(* IEC 61131-3 sources: beebread/doc (part 6) *)

// Commented out for beedance: it uses CODE, which is commented out.
// FUNCTION_BLOCK DNS_REV_CLIENT
// VAR_IN_OUT
// 	IP_C : IP_C; (* IP_Control management structure *)
// 	S_BUF : NETWORK_BUFFER;
// 	R_BUF : NETWORK_BUFFER;
// END_VAR
// VAR_INPUT
// 	ACTIVATE : BOOL;
// 	IP4 : DWORD;
// 	IP4_DNS : DWORD;
// END_VAR
// VAR_OUTPUT
// 	DOMAIN : STRING;
// 	DONE : BOOL;
// 	ERROR : DWORD;
// END_VAR
// VAR
// 	IP_FIFO : IP_FIFO;
// 	ip_state : BYTE;
// 	ip_id : BYTE;
// 	state : INT;
// 	ip4_copy : DWORD;
// 	d : STRING(27);
// 	activate_last : BOOL;
// 	i : INT;
// 	dl : INT;
// 	p1 : INT;
// 	char : BYTE;
// 	char_count : INT;
// 	tid : BYTE;
// END_VAR
//
// (* Domain Name System (query) *)
//
// CASE state OF
// 00: (* wait for rising edge on GET *)
// 	IF ACTIVATE AND NOT activate_last THEN
// 		ERROR := DWORD#0;
// 		ip4_copy := ip4; (* save IP4 *)
// 		ip_state := BYTE#1;
// 		DOMAIN := '';
// 		DONE := FALSE;
//
// 		d := '';
// 		FOR i := 1 TO 4 DO
// 			d := CONCAT(d,BYTE_TO_STRING(DWORD_TO_BYTE(IP4)));
// 			d := CONCAT(d,'.');
// 			IP4 := ROR(IP4,8);
// 		END_FOR;
// 		d := CONCAT(d,'in-addr.arpa');
// 		state := 10;
// 	END_IF;
//
// 10: (* register with IP_Control *)
// 	IF ip_state = BYTE#3 THEN
// 		dl := LEN(d);
//
// 		(* initialize send buffer *)
// 		char_count := 17 + dl;
// 		FOR i := 0 TO char_count DO
// 			S_BUF.BUFFER[i] := BYTE#00;
// 		END_FOR;
//
// 		tid := UINT_TO_BYTE(BYTE_TO_UINT(tid) + UINT#1);
// 		S_BUF.BUFFER[01] := tid; (* Transaction ID lowbyte *)
// 		S_BUF.BUFFER[02] := BYTE#16#01; (* Flags: highbyte *)
// 		S_BUF.BUFFER[05] := BYTE#16#01; (* Questions: lowbyte *)
//
// 		(* process the server name from back to front *)
// 		i := dl + 12;
// 		char_count := 0;
//
// 		WHILE i > 12 DO
// 			char := CODE(STR:=d,POS:=i - 12);
//
// 			(* check for main/sub domain name separator "." *)
// 			IF char = BYTE#46 THEN
// 				(* instead of the separator "." the length of the detected main/sub domain name is entered *)
// 				S_BUF.BUFFER[i] := INT_TO_BYTE(char_count);
// 				char_count := 0;
// 			ELSE
// 				S_BUF.BUFFER[i] := char; (* enter char into buffer *)
// 				char_count := char_count + 1; (* count number of chars *)
// 			END_IF;
// 			i := i - 1;
// 		END_WHILE;
//
// 		S_BUF.BUFFER[i] := INT_TO_BYTE(char_count); (* enter the length of the leftmost (first) domain name *)
// 		i := dl + 15; (* position after the server name *)
// 		S_BUF.BUFFER[i] := BYTE#12; (* Type: PTR (Domain name pointer) lowbyte *)
// 		i := i + 2;
// 		S_BUF.BUFFER[i] := BYTE#01; (* Class: IN lowbyte *)
// 		i := i + 1;
//
// 		(* set up IP data traffic *)
// 		IP_C.C_PORT := WORD#53; (* enter port number *)
// 		IP_C.C_IP := IP4_DNS; (* enter IP *)
// 		IP_C.C_MODE := BYTE#1; (* Mode: UDP+ACTIVE+PORT+IP *)
// 		IP_C.C_ENABLE := TRUE; (* enable connection setup *)
// 		IP_C.TIME_RESET := TRUE; (* reset timeout monitoring *)
// 		IP_C.R_OBSERVE  := TRUE; (* monitor data reception *)
// 		S_BUF.SIZE := INT_TO_UINT(i); (* enter send length *)
// 		R_BUF.SIZE := UINT#0; (* reset receive length *)
// 		state := 30;
// 	END_IF;
//
// 30:
// 	IF IP_C.ERROR <> DWORD#00 THEN
// 		ERROR := IP_C.ERROR;
// 	(* check whether the response telegram has the correct transaction ID and minimum length *)
// 	ELSIF (S_BUF.SIZE = UINT#0) AND (tid = R_BUF.BUFFER[1]) AND (R_BUF.SIZE >= INT_TO_UINT(i+12)) THEN
//
// 		(* check return code of the flags. 4 bits *)
// 		ERROR := BYTE_TO_DWORD(R_BUF.BUFFER[3] AND BYTE#2#0000_1111);
//
// 		IF ERROR = DWORD#00 THEN
//
// 			i := R_BUF.SIZE - 2;
// 			WHILE R_BUF.BUFFER[i] > 0 DO
// 				IF i = 0 THEN EXIT; END_IF;
// 				i := i - 1;
// 			END_WHILE;
//
// 			i := i + 2;
// 			p1 := i + 1;
// 			WHILE i < R_BUF.SIZE DO
// 				dl := R_BUF.BUFFER[i];
// 				IF dl > 0 THEN
// 					R_BUF.BUFFER[i] := BYTE#46;
// 					i := i + dl + 1;
// 				ELSE
// 					DOMAIN := BUFFER_TO_STRING(PT:=REF(R_BUF.BUFFER),SIZE:=SIZEOF(R_BUF.BUFFER),START:=p1,STOP:=i-1);
// 					EXIT;
// 				END_IF;
// 			END_WHILE;
// 			state := 0;
// 			DONE := TRUE;
// 		END_IF;
// 	END_IF;
//
// 	IF ERROR <> DWORD#0 THEN
// 		state := 0;
// 	END_IF;
//
// 	IF state = 0 THEN
// 		IP_C.R_OBSERVE := FALSE; (* monitor data reception *)
// 		ip_state := BYTE#4; (* unregister *)
// 	END_IF;
//
// END_CASE;
//
// activate_last := ACTIVATE; (* save last status for edge detection *)
//
// (* IP_FIFO *)
// IP_FIFO(FIFO:=IP_C.FIFO,STATE:=ip_state,ID:=ip_id);
//
// (*----------------------------------------------------------------------------------------------------------------*)
// (* Flags: 0x0100 (Standard query)                                                                                            *)
// (* 0... .... .... .... = Response: Message is a query                                                                   *)
// (* .000 0... ....  = Opcode: Standard query (0)                                                                          *)
// (* .... ..0. .... .... = Truncated: Message is not truncated                                                          *)
// (* .... ...1 .... .... = Recursion desired: Do query recursively                                                    *)
// (* .... .... .0.. .... = Z: reserved (0)                                                                                                  *)
// (* .... .... ...0 .... = Non-authenticated data OK: Non-authenticated data is unacceptable *)
// (*-----------------------------------------------------------------------------------------------------------------*)
//
// (*
// Errorcodes  Description	References
// 000	No error. 		 	The request completed successfully.
// 001	Format error. 		The name server was unable to interpret the query.
// 002	Server failure.  	The name server was unable to process this query due to a problem with the name server.
// 003	Name Error. 	 	Meaningful only for responses from an authoritative name server, this code signifies that the domain name referenced in the query does not exist.
// 004	Not Implemented. 	The name server does not support the requested kind of query.
// 005	Refused. 			The name server refuses to perform the specified operation for policy reasons.
//   						 For example, a name server may not wish to provide the information to the particular requester, or a name server may not wish to perform a particular operation (e.g., zone transfer) for particular data.
// 006	YXDomain.			Name Exists when it should not.
// 007	YXRRSet. RR			Set Exists when it should not.
// 008	NXRRSet. RR			Set that should exist does not.
// 009	NotAuth.			Server Not Authoritative for zone.
// 010	NotZone,			Name not contained in zone.
// 255	Timeout				No Response
// *)
// END_FUNCTION_BLOCK

// Commented out for beedance: it reads or writes the bytes of a STRING through a pointer; a beedance reference (REF_TO) refers to a whole variable of its type.
// FUNCTION ELEMENT_COUNT : INT
// VAR_INPUT
// 	SEP : BYTE;
// END_VAR
// VAR_IN_OUT
// 	ELEMENT : STRING(ELEMENT_LENGTH);
// END_VAR
// VAR
// 	pt : REF_TO ARRAY[1..ELEMENT_LENGTH] OF BYTE;
// 	l: INT;
// 	pos: INT;
// END_VAR
//
// IF ELEMENT = '' THEN
// 	ELEMENT_COUNT := 0;
// ELSE
// 	PT := REF(ELEMENT);
// 	ELEMENT_COUNT := 1;
// 	l := LEN(ELEMENT);
// 	FOR pos := 1 TO l DO
// 		IF pt^[pos] = SEP THEN ELEMENT_COUNT := ELEMENT_COUNT + 1; END_IF;
// 	END_FOR;
// END_IF;
// END_FUNCTION

// Commented out for beedance: it reads or writes the bytes of a STRING through a pointer; a beedance reference (REF_TO) refers to a whole variable of its type.
// FUNCTION ELEMENT_GET : STRING(ELEMENT_LENGTH)
// VAR_INPUT
// 	SEP : BYTE;
// 	POS : INT;
// END_VAR
// VAR_IN_OUT
// 	ELEMENT : STRING(ELEMENT_LENGTH);
// END_VAR
// VAR
// 	i : INT := 1;
// 	o : INT := 1;
// 	pt : REF_TO ARRAY[1..ELEMENT_LENGTH] OF BYTE;
// 	po : REF_TO ARRAY[1..ELEMENT_LENGTH] OF BYTE;
// 	cnt: INT;
// 	c: BYTE;
// END_VAR
//
// (* load pointers *)
// pt := REF(ELEMENT);
// po := REF(ELEMENT_GET);
//
// (* search for the n-th occurence of a separation character and store position in i *)
// WHILE (cnt < pos) AND (i < ELEMENT_LENGTH) AND (pt^[i] > 0) DO
// 	IF pt^[i] = sep THEN cnt := cnt + 1; END_IF;
// 	i := i + 1;
// END_WHILE;
//
// (* copy the list element to output *)
// IF i < ELEMENT_LENGTH THEN c := pt^[i]; END_IF;
// WHILE (c <> sep) AND (c > 0) AND (o < ELEMENT_LENGTH) AND (i < ELEMENT_LENGTH) DO
// 	po^[o] :=pt^[i];
// 	o := o + 1;
// 	i := i + 1;
// 	c := pt^[i];
// END_WHILE;
//
// (* terminate the output string *)
// po^[o] := 0;
// END_FUNCTION

FUNCTION_BLOCK FILE_BLOCK
VAR_IN_OUT
	MODE : BYTE;
	FILENAME : STRING;
	FSD : FILE_SERVER_DATA;
	PT : NETWORK_BUFFER;
END_VAR
VAR_INPUT
	POS : UDINT;
END_VAR
VAR_OUTPUT
	ERROR : BYTE;
	DATA : BYTE;
END_VAR
VAR
	step : INT;
	i : INT;
	data_start : UDINT;
	data_stop : UDINT;

END_VAR

CASE step OF
0:	IF MODE > 0 THEN
		ERROR := 0;
		IF FSD.FILE_OPEN AND (FSD.FILE_SIZE = 0 OR POS >= FSD.FILE_SIZE) THEN
			ERROR := 255;
			MODE := 0;
		ELSIF POS < data_start OR POS > data_stop OR NOT FSD.FILE_OPEN THEN (* reading data necessary *)
			FSD.FILENAME := FILENAME;
			FSD.MODE := 1; (* open + read *)
			FSD.OFFSET := POS;
			PT.SIZE := 65535; (* read maximum number *);
			data_start := 0;
			data_stop := 0;
			step := 10;
		ELSE (* data is present in the buffer *)
			i := UDINT_TO_INT(POS - data_start); (* calculate index *)
			DATA := PT.BUFFER[i];
			MODE := 0;
			(* ---------------------- Debug-Message ----------------------------*)
			(* -----------------------------------------------------------------*)
		END_IF;
	END_IF;

10:	IF FSD.MODE = 0 THEN (* command finished *)
		IF FSD.ERROR > 0 THEN
			ERROR := FSD.ERROR; (* output error *)
			MODE := 0;
		ELSE
			data_start := POS;
			data_stop := POS + UINT_TO_UDINT(PT.SIZE) - 1;
		END_IF;
		step := 0;
	END_IF;
END_CASE;
END_FUNCTION_BLOCK

FUNCTION FILE_PATH_SPLIT : BOOL
VAR_INPUT
	FILENAME : STRING(STRING_LENGTH);
END_VAR
VAR_IN_OUT
	X : FILE_PATH_DATA;
END_VAR
VAR
	b : INT;
	c : INT;
	d : STRING(1);
	p1 : INT;
	p2 : INT;
END_VAR

X.DRIVE := '';
X.DIRECTORY := '';
X.FILENAME := '';
c := LEN(FILENAME);
IF c = 0 THEN
	FILE_PATH_SPLIT := FALSE;
	RETURN;
END_IF;

FOR b := 1 TO c DO
	d := MID(FILENAME, 1, b);
	IF d = ':' THEN
		p1 := b;
	ELSIF d = '/' OR d = '\' THEN
		p2 := b;
	END_IF;
END_FOR;

IF p1 = 2 THEN
	X.DRIVE := LEFT(FILENAME,p1);
END_IF;

IF p2 > 0 AND p2 > p1 THEN
	X.DIRECTORY := MID(FILENAME,p2 - p1,p1+1); (* len , pos *)
END_IF;

X.FILENAME := RIGHT(FILENAME,c - MAX (p1,p2));
FILE_PATH_SPLIT := TRUE;
END_FUNCTION

FUNCTION_BLOCK FILE_SERVER
VAR_IN_OUT
	FSD : FILE_SERVER_DATA;
	PT : NETWORK_BUFFER;
END_VAR
VAR
	buf_size : UDINT;
	handle : UINT; (* Filehandle *)
	read_max_length : UDINT;(* maximum data length *)
	file_position : UDINT;(* current write/read pointer *)
	used_filename : STRING;(* current file name *)
	length_read : UDINT;
	write_length : UDINT;
	length_written : UDINT;
	open_handle : UINT;
	seek_position : UDINT;
	seek_mode : INT;
	seek_data : ARRAY[0..1] OF DINT;
	tell_position : UDINT;
	open_mode : DWORD;
	last_mode: BYTE;
	command : BYTE;
	error_code : BYTE;
	error : BOOL;
	file_change : BOOL;
	step : INT;
	X : FW_AdsRdWrt;
	tmpDW : UDINT;
	para : BOOL;
	FSR : FILE_SERVER_RUNTIME;

END_VAR

CASE step OF
0:
	IF FSD.MODE = LIMIT(1,FSD.MODE,5) THEN

		(* ---------------------- Debug-Message ----------------------------*)
		(* -----------------------------------------------------------------------------*)

		(* initialization *)
		X.sNetId := '';
		X.tTimeout := T#5s;
		X.nPort := 10000; (* AMSPORT_R3_SYSSERV *)

		buf_size := SIZEOF(PT.BUFFER);

		IF FSD.MODE = 4 THEN (* File_Remove *)
			IF handle > 0 THEN
				File_change := TRUE;
				step := 32000; (* execute File_Close *)
			ELSE
				step := 90; (* execute File_Remove *)
			END_IF;

		ELSIF FSD.MODE = 5 THEN (* File_Close *)
			step := 32000; (* execute File_Close *)

		ELSIF handle = 0 THEN (* MODE 1,2,3 *)
			step := 100; (* file must be opened first *)

		ELSE (* file is open *)
			IF used_filename = FSD.FILENAME AND FSD.MODE = last_mode THEN (* no mode change? *)
				step := 200; (* continue without open procedure *)
			ELSE
				step := 32000;
				File_change := TRUE;
			END_IF;
		END_IF;
	END_IF;

(* ----------------------------------- *)
090: (* File_Remove *)
	command := 7; (* File Remove *)
	step := 95;

095: (* File_Remove finished *)
	IF command = 0 THEN
		step := 30000; (* exit *)
	END_IF;
(* ----------------------------------- *)

100: (* File_Open *)
	IF FSD.MODE = 3 THEN (* Open_New + File Write *)
		open_mode := 16#0001_001A; (* PATH_GENERIC + WRITEPLUS + BINARY *)
	ELSE (* Mode 1 Open_Exist + File _Read / Mode 2 Open_Exist + File_Write *)
		open_mode := 16#0001_0019; (* PATH_GENERIC + READPLUS + BINARY *)
	END_IF;
	command := 1; (* FileOpen *)
	step := 105;

105: (* file open finished *)
	IF command = 0 THEN
		IF error THEN
			step := 30000; (* exit *)
		ELSE
			(* enter file data *)
			handle := open_handle;
			used_filename := FSD.FILENAME;
			file_position := UDINT#4294967295; (* 16#FFFF_FFFF -> maximum = unknown *)
			last_mode := FSD.MODE;
			step := 110;
		END_IF;
	END_IF;

110: (* File Seek *)
	command := 5; (* File-Seek *)
	seek_position := 0;
	seek_mode := 2; (* SEEK_END - Seek from the end of file *)
	step := 115;

115: (* file seek finished *)
	IF command = 0 THEN
		IF error THEN
			step := 30000; (* exit *)
		ELSE
			command := 6; (* start file tell *)
			step := 120;
		END_IF;
	END_IF;

120: (* file tell finished *)
	IF command = 0 THEN
		IF error THEN
			step := 30000; (* exit *)
		ELSE
			FSD.FILE_SIZE := tell_position; (* current file size *)
			FSD.FILE_OPEN := TRUE;
			step := 200;
		END_IF;
	END_IF;

200: (* File Seek *)
	IF FSD.OFFSET = UDINT#4294967294 THEN (* 16#FFFF_FFFE -> set pointer to end of file *)
		command := 5; (* File-Seek *)
		seek_position := FSD.FILE_SIZE;
		seek_mode := 0; (* Seek from beginning of file *)
		step := 210;
	ELSIF FSD.OFFSET > FSD.FILE_SIZE THEN (* check for valid offset setting *)
		error_code := 255;
		step := 30000; (* exit *)
	ELSIF FSD.OFFSET <> file_position THEN
		command := 5; (* File-Seek *)
		seek_position := FSD.OFFSET;
		seek_mode := 0; (* Seek from beginning of file *)
		step := 210;
	ELSE
		step := 300;
	END_IF;

210: (* File Seek *)
	IF command = 0 THEN
		file_position := seek_position;
		IF error THEN
			step := 30000; (* exit *)
		ELSE
			step := 300;
		END_IF;
	END_IF;

300: (* Read or Write ? *)
	IF FSD.MODE = 1 THEN
		step := 400; (* Read *)
	ELSE
		step := 500; (* Write *)
	END_IF;

400: (* File Read *)
	IF UINT_TO_UDINT(PT.SIZE) > buf_size THEN (* limit read length to buffer size *)
		read_max_length := buf_size;
	ELSE
		read_max_length := UINT_TO_UDINT(PT.SIZE);
	END_IF;

	IF read_max_length > buf_size THEN
		read_max_length := buf_size;  (* limit read length to buffer size *)
	END_IF;

	(* adjust read length to file length *)
	IF file_position + read_max_length > FSD.FILE_SIZE THEN
		read_max_length := FSD.FILE_SIZE - file_position;
	END_IF;

	IF read_max_length > 0 THEN
		command := 3; (* File_Read *)
		step := 410;
	ELSE
		PT.SIZE := UINT#0;
		step := 30000; (* exit *)
	END_IF;

410: (* File Read *)
	IF command = 0 THEN
		PT.SIZE := UDINT_TO_UINT(length_read);
		IF NOT Error THEN
			file_position := file_position + length_read; (* correct current File_Position *)
			FSD.OFFSET := file_position;
		END_IF;
		step := 30000; (* exit *)
	END_IF;

500: (* File Write *)
	IF UINT_TO_UDINT(PT.SIZE) > buf_size THEN (* limit write length to buffer size *)
		write_length := buf_size;
	ELSE
		write_length := UINT_TO_UDINT(PT.SIZE);
	END_IF;

	IF write_length > 0 THEN
		command := 4; (* File_Write *)
		step := 510;
	ELSE
		step := 30000; (* exit *)
	END_IF;

510:
	IF command = 0 THEN
		IF NOT Error THEN
			file_position := file_position + length_written; (* correct current File_Position *)
			FSD.OFFSET := file_position;
			IF file_position > FSD.FILE_SIZE THEN (* file has grown *)
				FSD.FILE_SIZE := file_position;
			END_IF;
		END_IF;
		step := 30000; (* exit *)
	END_IF;

 (* --------------------------------------------- *)

30000: (* command done *)
	FSD.MODE := 0;
	FSD.ERROR := error_code;
	step := 0;

	(* ---------------- Debug-Message -----------------------*)
	(* --------------------------------------------- *)

32000:
	IF handle > 0 THEN
		command := 2; (* execute File_Close *)
	END_IF;
	step := 32100;

32100:
	IF command = 0 THEN (* file close finished *)
		(* clear file data *)
		FSD.FILE_OPEN := FALSE;
		file_position := 0;
		FSD.FILE_SIZE := 0;
		FSD.OFFSET := 0;
		used_filename := '';
		handle := 0;

		(* File_Name changed on the fly? *)
		IF file_change THEN
			file_change := FALSE;
			step := 0;
		ELSE
			step := 30000;
		END_IF;
	END_IF;

END_CASE;

X(bExecute := FALSE); (* cyclic FW_AdsRdWrt call *)

FSR(MODE:=BYTE#0,COMMAND:=command,FSD:=FSD); (* monitor file server runtime / command start *)

(* ------------ File Open ------------- *)
IF command = 1 THEN
	IF NOT para THEN
		para := TRUE;
		X(	nIdxGrp := 120, (* SYSTEMSERVICE_FOPEN *)
			nidxOffs := open_mode,
			cbWriteLen := SIZEOF(FSD.FILENAME),
			pWriteBuff := REF(FSD.FILENAME),
			cbReadLen := SIZEOF(tmpDW),
			pReadBuff := REF(tmpDW),
			bExecute := TRUE
			);
	ELSIF X.bBusy = FALSE THEN
		para := FALSE;
		error := X.bError;
		error_code := SEL(error,0,UDINT_TO_BYTE(X.nErrId + 16#10));

		IF X.cbRead >= SIZEOF(tmpDW) THEN
			open_handle := UDINT_TO_UINT(tmpDW);
		ELSE
			open_handle := 0;
		END_IF;
		command := 0;
		FSR(MODE:=BYTE#1,COMMAND:=command,FSD:=FSD); (* monitor file server runtime / command stop *)
		(* ---------------- Debug-Message -----------------------*)
		(* -----------------------------------------------------------------*)
	END_IF;
END_IF;

(* ----------- File Close ------------- *)
IF command = 2 THEN
	IF NOT para THEN
		para := TRUE;
		X(	nIdxGrp := 121, (* SYSTEMSERVICE_FCLOSE *)
			nidxOffs := handle,
			cbWriteLen := 0,
			pWriteBuff := 0,
			cbReadLen := 0,
			pReadBuff := 0,
			bExecute := TRUE
			);
	ELSIF X.bBusy = FALSE THEN
		para := FALSE;
		error := X.bError;
		error_code := SEL(error,0,UDINT_TO_BYTE(X.nErrId + 16#30));
		command := 0;
		FSR(MODE:=BYTE#1,COMMAND:=command,FSD:=FSD); (* monitor file server runtime / command stop *)
		(* ---------------- Debug-Message -----------------------*)
		(* -----------------------------------------------------------------*)
	END_IF;
END_IF;

(* ------------ File Read ------------- *)
IF command = 3 THEN
	IF NOT para THEN
		para := TRUE;
		X(	nIdxGrp := 122, (* SYSTEMSERVICE_FREAD *)
			nidxOffs := handle,
			cbWriteLen := 0,
			pWriteBuff := 0,
			cbReadLen := read_max_length,
			pReadBuff := REF(PT.BUFFER),
			bExecute := TRUE
			);
	ELSIF X.bBusy = FALSE THEN
		length_read := X.cbRead;
		para := FALSE;
		error := X.bError;
		error_code := SEL(error,0,UDINT_TO_BYTE(X.nErrId + 16#40));
		command := 0;
		FSR(MODE:=BYTE#1,COMMAND:=command,FSD:=FSD); (* monitor file server runtime / command stop *)
		(* ---------------- Debug-Message -----------------------*)
		(* -----------------------------------------------------------------*)
	END_IF;
END_IF;

(* ------------ File Write ------------- *)
IF command = 4 THEN
	IF NOT para THEN
		para := TRUE;
		X(	nIdxGrp := 123, (* SYSTEMSERVICE_FWRITE *)
			nidxOffs := handle,
			cbWriteLen := write_length,
			pWriteBuff := REF(PT.BUFFER),
			cbReadLen := SIZEOF(length_written),
			pReadBuff := REF(length_written),
			bExecute := TRUE
			);
	ELSIF X.bBusy = FALSE THEN
		para := FALSE;
		error := X.bError;
		error_code := SEL(error,0,UDINT_TO_BYTE(X.nErrId + 16#50));
		command := 0;
		FSR(MODE:=BYTE#1,COMMAND:=command,FSD:=FSD); (* monitor file server runtime / command stop *)
		(* ---------------- Debug-Message -----------------------*)
		(* -----------------------------------------------------------------*)
	END_IF;
END_IF;

(* ------------ File Seek ------------- *)
IF command = 5 THEN
	IF NOT para THEN
		para := TRUE;
		seek_data[0] := UDINT_TO_DINT(seek_position);
		seek_data[1] := INT_TO_DINT(seek_mode);

		X(	nIdxGrp := 124, (* SYSTEMSERVICE_FSEEK *)
			nidxOffs := handle,
			cbWriteLen := SIZEOF(seek_data),
			pWriteBuff := REF(seek_data),
			cbReadLen := 0,
			pReadBuff := 0,
			bExecute := TRUE
			);
	ELSIF X.bBusy = FALSE THEN
		para := FALSE;
		error := X.bError;
		error_code := SEL(error,0,UDINT_TO_BYTE(X.nErrId + 16#60));
		command := 0;
		FSR(MODE:=BYTE#1,COMMAND:=command,FSD:=FSD); (* monitor file server runtime / command stop *)
		(* ---------------- Debug-Message -----------------------*)
		(* -----------------------------------------------------------------*)
	END_IF;
END_IF;

(* ------------ File Tell ------------- *)
IF command = 6 THEN
	IF NOT para THEN
		para := TRUE;
		X(	nIdxGrp := 125, (* SYSTEMSERVICE_FTELL *)
			nidxOffs := handle,
			cbWriteLen := 0,
			pWriteBuff := 0,
			cbReadLen := SIZEOF(tell_position),
			pReadBuff := REF(tell_position),
			bExecute := TRUE
			);
	ELSIF X.bBusy = FALSE THEN
		para := FALSE;
		error := X.bError;
		error_code := SEL(error,0,UDINT_TO_BYTE(X.nErrId + 16#70));
		command := 0;
		FSR(MODE:=BYTE#1,COMMAND:=command,FSD:=FSD); (* monitor file server runtime / command stop *)
		(* ---------------- Debug-Message -----------------------*)
		(* -----------------------------------------------------------------*)
	END_IF;
END_IF;

(* ------------ File Remove ------------- *)
IF command = 7 THEN
	IF NOT para THEN
		para := TRUE;
		X(	nIdxGrp := 131, (* SYSTEMSERVICE_FDELETE *)
			nidxOffs := 16#0001_0000, (* PATH_GENERIC *)
			cbWriteLen := SIZEOF(FSD.FILENAME),
			pWriteBuff := REF(FSD.FILENAME),
			cbReadLen := 0,
			pReadBuff := 0,
			bExecute := TRUE
			);
	ELSIF X.bBusy = FALSE THEN
		para := FALSE;
		error := X.bError;
		error_code := SEL(error,0,UDINT_TO_BYTE(X.nErrId + 16#80));
		command := 0;
		FSR(MODE:=BYTE#1,COMMAND:=command,FSD:=FSD); (* monitor file server runtime / command stop *)
		(* ---------------- Debug-Message -----------------------*)
		(* -----------------------------------------------------------------*)
	END_IF;
END_IF;

(* ---------------- Debug-Message -----------------------*)
(* -----------------------------------------------------------------*)
END_FUNCTION_BLOCK

FUNCTION_BLOCK FILE_SERVER_RUNTIME
VAR_INPUT
	MODE : BYTE;
	COMMAND : BYTE;
END_VAR
VAR_IN_OUT
	FSD : FILE_SERVER_DATA;
END_VAR
VAR
	last_command : BYTE;
	init : BOOL;
	start_tx : DWORD;
	stop_tx : DWORD;
	runtime : DWORD;
END_VAR

IF init = FALSE THEN
	init := TRUE;
	FSD.RUNTIME.TIME_FILE_OPEN_MIN := UDINT#99999999;
	FSD.RUNTIME.TIME_FILE_CLOSE_MIN := UDINT#99999999;
	FSD.RUNTIME.TIME_FILE_READ_MIN := UDINT#99999999;
	FSD.RUNTIME.TIME_FILE_WRITE_MIN := UDINT#99999999;
	FSD.RUNTIME.TIME_FILE_TELL_MIN := UDINT#99999999;
	FSD.RUNTIME.TIME_FILE_SEEK_MIN := UDINT#99999999;
	FSD.RUNTIME.TIME_FILE_DELETE_MIN := UDINT#99999999;
END_IF;

(* wait for File_Server command *)
IF MODE = BYTE#0 THEN

	(* new command detected *)
	IF last_command = BYTE#0 AND COMMAND <> BYTE#0 THEN

		(* read system time *)
		start_tx := T_PLC_MS();

	END_IF;
END_IF;

IF MODE = BYTE#1 THEN

	(* read system time *)
	stop_tx:=  T_PLC_MS();

	runtime:= (stop_tx - start_tx);

	CASE BYTE_TO_INT(COMMAND) OF

	1:	FSD.RUNTIME.TIME_FILE_OPEN_CUR := runtime; 			(* current runtime *)
		IF FSD.RUNTIME.TIME_FILE_OPEN_MAX < runtime THEN
			FSD.RUNTIME.TIME_FILE_OPEN_MAX := runtime;		(* new max runtime *)
		END_IF;
		IF FSD.RUNTIME.TIME_FILE_OPEN_MIN > runtime THEN
			FSD.RUNTIME.TIME_FILE_OPEN_MIN := runtime;		(* new min runtime *)
		END_IF;

	2:	FSD.RUNTIME.TIME_FILE_CLOSE_CUR := runtime; 			(* current runtime *)
		IF FSD.RUNTIME.TIME_FILE_CLOSE_MAX < runtime THEN
			FSD.RUNTIME.TIME_FILE_CLOSE_MAX := runtime;		(* new max runtime *)
		END_IF;
		IF FSD.RUNTIME.TIME_FILE_CLOSE_MIN > runtime THEN
			FSD.RUNTIME.TIME_FILE_CLOSE_MIN := runtime;		(* new min runtime *)
		END_IF;

	3:	FSD.RUNTIME.TIME_FILE_READ_CUR := runtime; 			(* current runtime *)
		IF FSD.RUNTIME.TIME_FILE_READ_MAX < runtime THEN
			FSD.RUNTIME.TIME_FILE_READ_MAX := runtime;		(* new max runtime *)
		END_IF;
		IF FSD.RUNTIME.TIME_FILE_READ_MIN > runtime THEN
			FSD.RUNTIME.TIME_FILE_READ_MIN := runtime;		(* new min runtime *)
		END_IF;

	4:	FSD.RUNTIME.TIME_FILE_WRITE_CUR := runtime; 			(* current runtime *)
		IF FSD.RUNTIME.TIME_FILE_WRITE_MAX < runtime THEN
			FSD.RUNTIME.TIME_FILE_WRITE_MAX := runtime;		(* new max runtime *)
		END_IF;
		IF FSD.RUNTIME.TIME_FILE_WRITE_MIN > runtime THEN
			FSD.RUNTIME.TIME_FILE_WRITE_MIN := runtime;		(* new min runtime *)
		END_IF;

	5:	FSD.RUNTIME.TIME_FILE_SEEK_CUR := runtime; 			(* current runtime *)
		IF FSD.RUNTIME.TIME_FILE_SEEK_MAX < runtime THEN
			FSD.RUNTIME.TIME_FILE_SEEK_MAX := runtime;		(* new max runtime *)
		END_IF;
		IF FSD.RUNTIME.TIME_FILE_SEEK_MIN > runtime THEN
			FSD.RUNTIME.TIME_FILE_SEEK_MIN := runtime;		(* new min runtime *)
		END_IF;

	6:	FSD.RUNTIME.TIME_FILE_TELL_CUR := runtime; 			(* current runtime *)
		IF FSD.RUNTIME.TIME_FILE_TELL_MAX < runtime THEN
			FSD.RUNTIME.TIME_FILE_TELL_MAX := runtime;		(* new max runtime *)
		END_IF;
		IF FSD.RUNTIME.TIME_FILE_TELL_MIN > runtime THEN
			FSD.RUNTIME.TIME_FILE_TELL_MIN := runtime;		(* new min runtime *)
		END_IF;

	7:	FSD.RUNTIME.TIME_FILE_DELETE_CUR := runtime; 			(* current runtime *)
		IF FSD.RUNTIME.TIME_FILE_DELETE_MAX < runtime THEN
			FSD.RUNTIME.TIME_FILE_DELETE_MAX := runtime;		(* new max runtime *)
		END_IF;
		IF FSD.RUNTIME.TIME_FILE_DELETE_MIN > runtime THEN
			FSD.RUNTIME.TIME_FILE_DELETE_MIN := runtime;		(* new min runtime *)
		END_IF;

	END_CASE;

END_IF;

last_command := COMMAND;
END_FUNCTION_BLOCK

// Commented out for beedance: it has a comment between UNTIL and END_REPEAT, which beedance does not parse yet.
// FUNCTION_BLOCK FTP_CLIENT
// VAR_INPUT
// 	ACTIVATE : BOOL;
// 	FILENAME : STRING;
// 	FTP_URL : STRING(STRING_LENGTH);
// 	FTP_DOWNLOAD : BOOL;
// 	FTP_ACTIV : BOOL;
// 	FILE_DELETE : BOOL;
// 	TIMEOUT : TIME;
// 	DNS_IP4 : DWORD;
// 	PLC_IP4 : DWORD;
// END_VAR
// VAR_OUTPUT
// 	DONE : BOOL;
// 	BUSY : BOOL;
// 	ERROR_C : DWORD;
// 	ERROR_T : BYTE;
// END_VAR
// VAR
// 	IP_C1 : IP_C; (* IP_Control management structure *)
// 	IP_C2 : IP_C; (* IP_Control management structure *)
// 	S_BUF1 : NETWORK_BUFFER;
// 	S_BUF2 : NETWORK_BUFFER;
// 	R_BUF1 : NETWORK_BUFFER;
// 	R_BUF2 : NETWORK_BUFFER;
// 	URL_DATA : url;
// 	DNS_CLIENT : DNS_CLIENT;
// 	IPC1 : IP_CONTROL;
// 	IPC2 : IP_CONTROL;
// 	FS : FILE_SERVER;
// 	FSD : FILE_SERVER_DATA;
//
// 	activate_last : BOOL;
// 	step : INT;
// 	snd_step : INT;
// 	snd_text :	STRING(STRING_LENGTH);
// 	rcv_text :	STRING(STRING_LENGTH);
// 	rcv_state : INT;
// 	TON_WAIT : TON;
// 	last_step : INT;
// 	next_step : INT;
// 	idx1 : INT;
// 	idx2 : INT;
// 	str1 : STRING(STRING_LENGTH);
// 	str2 : STRING(STRING_LENGTH);
// 	ftp_path : STRING;
// 	byar : ARRAY [0..5] OF BYTE;
// 	dw_tmp : DWORD;
// 	w_tmp : WORD;
// 	fpd : FILE_PATH_DATA;
// 	timeout2 : TIME;
// 	timeout3 : TIME;
// 	ftp_file_size : UDINT;
// 	ip_c1_red_disable : BOOL; (* IP_CONTROL 1 - suppress remote disconnect error *)
// 	ip_c2_red_disable : BOOL; (* IP_CONTROL 1 - suppress remote disconnect error *)
//
// 	(*LOG_MSG : LOG_MSG;
// 	_debug_enable : BOOL := FALSE;*)
//
// END_VAR
// CASE step OF
//
// 00:	IF ACTIVATE AND NOT activate_last THEN
// 		ftp_file_size := UDINT#0;
// 		TIMEOUT := MAX(T#10s,TIMEOUT);
// 		timeout2 := TIMEOUT + T#1s;
// 		timeout3 := TIMEOUT / 2;
// 		DONE := FALSE;
// 		ip_c1_red_disable := FALSE;
// 		ip_c2_red_disable := FALSE;
// 		ERROR_C := DWORD#0;
// 		ERROR_T := BYTE#0;
// 		FSD.ERROR := BYTE#0;
// 		URL_DATA := STRING_TO_URL(STR:=FTP_URL,DEFAULT_PROTOCOL:='',DEFAULT_PATH:='/');
// 		IF LEN(URL_DATA.USER) = 0 THEN
// 			URL_DATA.USER := 'Anonymous';
// 			URL_DATA.PASSWORD := 'User@';
// 		END_IF;
//
// 		FILE_PATH_SPLIT(FILENAME:=FILENAME,X:=fpd); (* split file path *)
// 		str1 := fpd.FILENAME; (* buffer temporarily *)
// 		FILE_PATH_SPLIT(FILENAME:=URL_DATA.PATH,X:=fpd); (* split FTP path *)
// 		IF LEN(fpd.FILENAME) = 0 THEN (* if the FTP path contains no file name, use the name of the local file *)
// 			ftp_path := CONCAT(URL_DATA.PATH,str1);
// 		ELSE
// 			ftp_path := URL_DATA.PATH;
// 		END_IF;
// 		step := 10;
// 	END_IF;
//
// 10:	IF DNS_CLIENT.DONE THEN
// 		step := 20;
// 	ELSIF DNS_CLIENT.ERROR <> DWORD#0 THEN
// 		ERROR_C := DNS_CLIENT.ERROR;
// 		ERROR_T := BYTE#1;
// 		step := 980;
// 	END_IF;
//
// 20:	(* set up FTP control channel *)
// 	IP_C1.C_PORT := WORD#21; (* enter port number *)
//   	IP_C1.C_IP := DNS_CLIENT.IP4; (* enter IP *)
//   	IP_C1.C_MODE := BYTE#0; (* Mode: TCP+ACTIV+PORT *)
//   	IP_C1.TIME_RESET := TRUE; (* reset timeout monitoring *)
//   	IP_C1.C_ENABLE := TRUE; (* enable connection setup *)
//   	IP_C1.R_OBSERVE := TRUE; (* receive monitoring *)
// 	R_BUF1.SIZE := UINT#0;
//
//   	IP_C2.C_ENABLE   := FALSE; (* block connection setup *)
// 	step := 30;
//
// 30:	IF rcv_state = 220 THEN (* 220 = Service ready for new user *)
// 		snd_text := CONCAT('USER ',URL_DATA.USER);
// 		next_step := 40;
// 	END_IF;
//
// 40:	IF rcv_state = 331 THEN (* 331 = User name okay, need password *)
// 		snd_text := CONCAT('PASS ',URL_DATA.PASSWORD);
// 		next_step := 50;
// 	ELSIF rcv_state = 230 THEN (* 230 = User logged in, proceed *)
// 		next_step := 50;
// 	ELSIF rcv_state = 220 THEN (* 220 = Service ready for new user *)
// 		next_step := 20; (* WORK connection should be closed/opened *)
// 	END_IF;
//
// 50:	IF rcv_state = 230 THEN (* 230 = User logged in, proceed *)
// 		snd_text := 'TYPE I';  (* activate binary mode *)
// 		next_step := 54;
// 	END_IF;
//
// 54:	IF rcv_state = 200 THEN (* 200 = Command okay *)
// 		IF FTP_DOWNLOAD THEN (* receive file from FTP *)
// 			snd_text := CONCAT('SIZE ', ftp_path); (* SIZE /PATH/FILENAME *)
// 			next_step := 56;
// 		ELSE
// 			step := 60;
// 		END_IF;
// 	END_IF;
//
// 56:	IF rcv_state = 213 THEN (* 213 Filesize *)
// 		str1 := ELEMENT_GET(SEP:=BYTE#32,POS:=1,ELEMENT:=rcv_text);
// 		ftp_file_size := STRING_TO_UDINT(str1); (* determine file size in bytes *)
// 		step := 60;
// 	END_IF;
//
// 60:	IF FTP_ACTIV THEN (* FTP server active *)
// 		IF URL_DATA.PORT = WORD#0 THEN
// 			URL_DATA.PORT := WORD#20; (* default data channel *)
// 		END_IF;
// 		str2 := '';
// 		dw_tmp := PLC_IP4;
// 		FOR idx1 := 0 TO 5 DO
// 			IF idx1 = 4 THEN
// 				dw_tmp := ROR(WORD_TO_DWORD(URL_DATA.PORT),8);
// 			ELSE
// 				dw_tmp := ROL(dw_tmp,8);
// 			END_IF;
// 			str2 := CONCAT(str2,BYTE_TO_STRING(DWORD_TO_BYTE(dw_tmp)));
// 			IF idx1 < 5 THEN
// 				str2 := CONCAT(str2,',');
// 			END_IF;
// 		END_FOR;
// 		dw_tmp := DNS_CLIENT.IP4; (* enter IP *)
// 		w_tmp := URL_DATA.PORT; (* port number of the data channel *)
// 		snd_text := CONCAT('PORT ',str2); (* switch FTP server to active mode *)
// 		next_step := 80;
// 	ELSE
// 		snd_text := 'PASV';  (* switch FTP server to passive mode *)
// 		next_step := 70;
// 	END_IF;
// 	step := 999; (* wait for next_step *)
//
// 70:	IF rcv_state = 227 THEN (* 227 = Entered Passive Mode (213,202,225,43,212,186) *)
// 		idx1 := FIND(rcv_text , '(' );
// 		idx2 := FIND(rcv_text , ')' );
// 		IF idx1 > 0 AND idx2 > idx1+1 THEN
// 			str1 := MID(rcv_text, idx2 - idx1 - 1, idx1+1);
// 			FOR idx1 := 0 TO 5 DO
// 				str2 := ELEMENT_GET(SEP:=BYTE#44,POS:=idx1,ELEMENT:=str1);
// 				byar[idx1] := STRING_TO_BYTE(str2);
// 			END_FOR;
// 			dw_tmp := DWORD_OF_BYTE(byar[0],byar[1],byar[2],byar[3]); (* IP address of the data channel *)
// 			w_tmp := WORD_OF_BYTE(byar[4],byar[5]); (* port number of the data channel *)
// 		END_IF;
// 		step := 100;
// 	END_IF;
//
// 80:	IF rcv_state = 200 THEN (* 200 = PORT command successful *)
// 		step := 100;
// 	END_IF;
//
// 100:IP_C2.C_MODE := SEL(FTP_ACTIV,BYTE#0,BYTE#2); (* active = mode 2: TCP+PASSIVE+PORT / passive = mode 0: TCP+ACTIVE+PORT *)
// 	IP_C2.C_IP := dw_tmp; (* IP address of the data channel *)
// 	IP_C2.C_PORT := w_tmp; (* port number of the data channel *)
//   	IP_C2.TIME_RESET := TRUE; (* reset timeout monitoring *)
//   	IP_C2.C_ENABLE := TRUE; (* enable connection setup *)
// 	IP_C2.R_OBSERVE := FALSE; (* receive monitoring *)
// 	R_BUF2.SIZE := UINT#0;
// 	step := 120;
//
// 120:IF IP_C2.C_STATE > BYTE#127 THEN (* FTP data channel established *)
// 		IF FTP_DOWNLOAD THEN (* receive file from FTP *)
// 			IP_C2.MAILBOX[3] := BYTE#1; (* block IP receive *)
// 			step := 400;
// 		ELSE
// 			snd_text := 'STOR ';
// 			next_step := 140;
// 			snd_text := CONCAT(snd_text, ftp_path); (* STORE /PATH/FILENAME *)
// 			step := 999; (* wait for next_step *)
// 		END_IF;
// 	END_IF;
//
// (* ============== send file to FTP ================ *)
//
// 140:IF rcv_state = 125 OR rcv_state = 150 THEN (* 125 = Data connection already open / 150 = File status okay; about to open data connection *)
// 		step := 160;
// 	END_IF;
//
// 160:FSD.FILENAME := FILENAME; (* file name *)
// 	FSD.MODE := BYTE#1; (* open existing file for reading *)
// 	FSD.OFFSET := UDINT#0; (* start at beginning of file *)
// 	S_BUF2.SIZE := UINT#65535; (* read maximum length *)
// 	IP_C2.MAILBOX[2] := BYTE#1; (* block IP send *)
// 	step := 200;
//
// 200:IF FSD.MODE = BYTE#0 AND FSD.ERROR = BYTE#0 THEN
// 		IP_C2.MAILBOX[2] := BYTE#0; (* allow IP send *)
// 		step := 210;
// 	END_IF;
//
// 210:IF S_BUF2.SIZE = UINT#0 THEN (* wait until all data is sent *)
// 		IF FSD.FILE_SIZE - FSD.OFFSET > UDINT#0 THEN
// 			FSD.MODE := BYTE#1; (* open existing file for reading *)
// 			S_BUF2.SIZE := UINT#65535; (* read maximum length *)
// 			IP_C2.MAILBOX[2] := BYTE#1; (* block IP send *)
// 			step := 200;
// 		ELSE
// 			IP_C2.C_ENABLE := FALSE; (* close FTP data channel *)
// 			step := 300;
// 		END_IF;
// 	END_IF;
//
// 300:IF rcv_state = 226 THEN (* 226 Closing data connection. Requested file action successful  *)
// 		snd_text := 'QUIT';
// 		ip_c1_red_disable := TRUE;
// 		next_step := 320;
// 	END_IF;
//
// 320:IF rcv_state = 221 OR TON_WAIT.ET > timeout3  THEN (* 221 Service closing control connection *)
// 		IP_C1.C_ENABLE := FALSE; (* close FTP control channel *)
// 		IF FILE_DELETE THEN (* delete file after transfer *)
// 			FSD.MODE := BYTE#4; (* File Remove *)
// 			step := 340;
// 		ELSE
// 			step := 900;
// 		END_IF;
// 	END_IF;
//
// 340:IF FSD.MODE = BYTE#0 AND FSD.ERROR = BYTE#0 THEN
// 		step := 900;
// 	END_IF;
//
// (*  ============== receive file from FTP  ============== *)
//
// 400:snd_text := 'RETR ';
// 	next_step := 410;
// 	snd_text := CONCAT(snd_text, ftp_path); (* RETR /PATH/FILENAME *)
// 	step := 999; (* wait for next_step *)
//
// 410:IF rcv_state = 125 OR rcv_state = 150 THEN (* 125 = Data connection already open / 150 = File status okay; about to open data connection *)
// 		IP_C2.R_OBSERVE := TRUE; (* receive monitoring *)
// 		step := 420;
// 	END_IF;
//
// 420:FSD.FILENAME := FILENAME; (* file name *)
// 	FSD.MODE := BYTE#3; (* create new file *)
// 	FSD.OFFSET := UDINT#0; (* start at beginning of file *)
// 	step := 460;
//
// 440:IF R_BUF2.SIZE > UINT#0 THEN (* wait until data has been received *)
// 		IP_C2.MAILBOX[3] := BYTE#1; (* block IP receive until data has been written to file *)
// 		FSD.MODE := BYTE#3; (* write data to file *)
// 		step := 460;
// 	ELSIF FSD.FILE_SIZE = ftp_file_size THEN (* connection closed?, or 226 = Closing data connection. Requested file action successful *)
// 		IP_C2.C_ENABLE := FALSE; (* close FTP data channel *)
// 		ip_c2_red_disable := TRUE;
// 		step := 700;
// 	END_IF;
//
// 460:IF FSD.MODE = BYTE#0 AND FSD.ERROR = BYTE#0 THEN (* wait until data has been written *)
// 		R_BUF2.SIZE := UINT#0; (* delete data *)
// 		IP_C2.MAILBOX[3] := BYTE#0; (* allow IP receive again *)
// 		step := 440;
// 	END_IF;
//
// (* ================================================== *)
//
// 700:IF rcv_state = 226 OR  TON_WAIT.ET > timeout3 THEN (* 226 Closing control connection. Requested file action successful  *)
// 		IF FTP_DOWNLOAD AND FILE_DELETE THEN (* FTP download and delete file? *)
// 			snd_text := CONCAT('DELE ', ftp_path); (* DELE /PATH/FILENAME *)
// 			next_step := 720;
// 		ELSE
// 			step := 740;
// 		END_IF;
// 	END_IF;
//
// 720:IF rcv_state = 250 THEN (* 250 Requested file action okay, completed *)
// 		step := 740;
// 	END_IF;
//
// 740:snd_text := 'QUIT';
// 	ip_c1_red_disable := TRUE;
// 	next_step := 760;
// 	step := 999; (* wait for next_step *)
//
// 760:IF rcv_state = 221 OR TON_WAIT.ET > timeout3 THEN (* 221 Service closing control connection  *)
// 		IP_C1.C_ENABLE := FALSE; (* close FTP control channel *)
// 		IF NOT FTP_DOWNLOAD AND FILE_DELETE THEN (* FTP upload and delete file after transfer *)
// 			FSD.MODE := BYTE#4; (* File Remove *)
// 			step := 780;
// 		ELSE
// 			step := 900;
// 		END_IF;
// 	END_IF;
//
// 780:IF FSD.MODE = BYTE#0 AND FSD.ERROR = BYTE#0 THEN
// 		step := 900;
// 	END_IF;
//
// (* ================================================== *)
//
// 900:DONE := TRUE;
// 	step := 980;
//
// 980:IP_C1.C_ENABLE := FALSE; (* close FTP control channel *)
// 	IP_C2.C_ENABLE := FALSE; (* close FTP data channel *)
// 	IP_C2.MAILBOX[2] := BYTE#0; (* allow IP send again *)
// 	IP_C2.MAILBOX[3] := BYTE#0; (* allow IP receive again *)
// 	S_BUF1.SIZE := UINT#0;
// 	S_BUF2.SIZE := UINT#0;
// 	R_BUF1.SIZE := UINT#0;
// 	R_BUF2.SIZE := UINT#0;
// 	ftp_file_size := UDINT#0;
// 	snd_step := 0;
// 	next_step := 0;
// 	FSD.MODE := BYTE#5; (* close file *)
// 	step := 990;
//
// 990:IF IP_C1.C_STATE = BYTE#0 AND IP_C2.C_STATE = BYTE#0 AND FSD.FILE_OPEN = FALSE THEN
// 		step := 0;
// 	END_IF;
//
// 999: ; (* dummy step, wait until a new step becomes active through "next_step" *)
//
// END_CASE;
//
// (* ++++++++++++++++++++++++++++++++++++++++++++++++++++++++++ *)
//
// IF step >= 30 THEN
// 	IF R_BUF1.SIZE > UINT#0 THEN (* data received? *)
// 		idx1 := UINT_TO_INT(R_BUF1.SIZE);
// 		REPEAT (* detect line termination and determine real end of TEXT *)
// 			idx1 := idx1 - 1;
// 		UNTIL idx1 = 0 OR R_BUF1.BUFFER[idx1] >= BYTE#32 (* TRUE = EXIT *)
// 		END_REPEAT;
// 		idx1 := idx1 + 1; (* convert index to SIZE *)
// 		rcv_text := BUFFER_TO_STRING(PT:=REF(R_BUF1.BUFFER),SIZE:=idx1,START:=0,STOP:=STRING_LENGTH-1);
// 		IF LEN(rcv_text) >= 3 THEN (* check and evaluate status code *)
// 			str1 := LEFT(rcv_text,3);
// 			IF IS_NUM(STR:=str1) THEN (* contains only digits? *)
// 				rcv_state := STRING_TO_INT(str1);
// 			END_IF;
// 			IP_C1.R_OBSERVE := FALSE;
// 		END_IF;
// 		R_BUF1.SIZE := UINT#0; (* delete data *)
//
// 	        (*####################  DEBUG-MESSAGE  ###################################*)
// 	        (*IF _debug_enable THEN
// 	          LOG_CL.NEW_MSG := 'RCV: >~1<';
// 	          LOG_CL.PRINTF[1] := rcv_text;
// 	          LOG_MSG();
// 	        END_IF;*)
// 	        (*########################################################################*)
//
// 	END_IF;
// END_IF;
//
// (* automatic data sending *)
//
// CASE snd_step OF
//
// 00:	IF LEN(snd_text) > 0 THEN
// 	        (*####################  DEBUG-MESSAGE  ###################################*)
// 	        (*IF _debug_enable THEN
// 	          LOG_CL.NEW_MSG := 'SND: >~1<';
// 	          LOG_CL.PRINTF[1] := snd_text;
// 	          LOG_MSG();
// 	        END_IF;*)
// 	        (*########################################################################*)
// 		_STRING_TO_BUFFER(str:=snd_text,pos:=0,pt:=REF(S_BUF1.BUFFER),size:=SIZEOF(S_BUF1.BUFFER)); (* copy string into buffer *)
// 		idx1 := LEN(snd_text);
// 		S_BUF1.BUFFER[idx1] := BYTE#16#0D;
// 		idx1 := idx1 + 1;
// 		S_BUF1.BUFFER[idx1] := BYTE#16#0A;
// 		idx1 := idx1 + 1;
// 		S_BUF1.SIZE := INT_TO_UINT(idx1); (* enter send length *)
// 		R_BUF1.SIZE := UINT#0; (* reset receive buffer *)
// 		IP_C1.R_OBSERVE := TRUE;
// 		rcv_state := 9999; (* clear last FTP status *)
// 		snd_text := '';
// 		snd_step := 10;
// 	END_IF;
//
// 10:	IF S_BUF1.SIZE = UINT#0 THEN (* wait until all data is sent *)
// 		step := next_step;
// 		snd_step := 0;
// 	END_IF;
//
// END_CASE;
//
// (* global error handling for main routine *)
// IF ERROR_T = BYTE#0 AND step > 20 THEN (* no error stored yet and main routine active *)
//
// 	IF IP_C1.ERROR > DWORD#0 AND IP_C1.C_ENABLE AND NOT IP_C1.TIME_RESET THEN  (* IP Control 1 *)
// 		IF ip_c1_red_disable = FALSE OR IP_C1.ERROR <> DWORD#16#FD000000 THEN
// 			ERROR_C := IP_C1.ERROR;
// 			ERROR_T := BYTE#2;
// 			step := 980;
// 		END_IF;
// 	END_IF;
//
// 	IF IP_C2.ERROR > DWORD#0 AND IP_C2.C_ENABLE AND NOT IP_C2.TIME_RESET THEN  (* IP Control 2 *)
// 		IF ip_c2_red_disable = FALSE OR IP_C2.ERROR <> DWORD#16#FD000000 THEN
// 			ERROR_C := IP_C2.ERROR;
// 			ERROR_T := BYTE#3;
// 			step := 980;
// 		END_IF;
// 	END_IF;
//
// 	IF FSD.MODE = BYTE#0 THEN
// 		IF FSD.ERROR > BYTE#0 THEN
// 			ERROR_C := BYTE_TO_DWORD(FSD.ERROR);
// 			ERROR_T := BYTE#4; (* file access *)
// 			step := 980;
// 		END_IF;
// 	END_IF;
// END_IF;
//
// IF TON_WAIT.Q THEN (* sequence fault - step chain *)
// 	ERROR_C := SHL(INT_TO_DWORD(step),16) OR INT_TO_DWORD(rcv_state); (* enter current step and last FTP status *)
// 	ERROR_T := BYTE#5;
// 	step := 980;
// END_IF;
//
// (* ######################################################## *)
//
// DNS_CLIENT(IP_C:=IP_C1, S_BUF:=S_BUF1, R_BUF:=R_BUF1, DOMAIN:=URL_DATA.DOMAIN, IP4_DNS:= DNS_IP4, ACTIVATE:=step=10); (* DNS-Client *)
// IPC1(IP:= DWORD#0, PORT:= WORD#0 , TIME_OUT:= TIMEOUT, IP_C:= IP_C1, S_BUF:= S_BUF1, R_BUF:= R_BUF1); (* FTP control channel *)
// IPC2(IP:= DWORD#0, PORT:= WORD#0 , TIME_OUT:= TIMEOUT, IP_C:= IP_C2, S_BUF:= S_BUF2, R_BUF:= R_BUF2); (* FTP data channel *)
//
// TON_WAIT(IN:=step = last_step AND step > 0,PT:=timeout2);
// last_step := step;
// activate_last := ACTIVATE;
// BUSY := step <> 0;
//
// IF FTP_DOWNLOAD THEN (* FILE_SERVER *)
// 	FS(FSD:=FSD,PT:=R_BUF2); (* receive file from FTP *)
// ELSE
// 	FS(FSD:=FSD,PT:=S_BUF2); (* send file to FTP *)
// END_IF;
// END_FUNCTION_BLOCK

// Commented out for beedance: it uses CHR_TO_STRING, which is commented out.
// FUNCTION_BLOCK GET_WAN_IP
// VAR_IN_OUT
// 	IP_C : IP_C; (* IP_Control management structure *)
// 	S_BUF : NETWORK_BUFFER;
// 	R_BUF : NETWORK_BUFFER;
// END_VAR
// VAR_INPUT
// 	ACTIVATE : BOOL;
// END_VAR
// VAR_OUTPUT
// 	WAN_IP4 : DWORD;
// 	DONE : BOOL;
// 	NEW_IP4 : BOOL;
// 	ERROR_C : DWORD;
// 	ERROR_T : BYTE;
// END_VAR
// VAR
// 	URL_DATA : url;
// 	DNS_CLIENT : DNS_CLIENT;
// 	HTTP_GET : HTTP_GET;
// 	activate_last : BOOL;
// 	wan_ip4_last : DWORD;
// 	state : INT;
// 	st_ip : STRING(120);
// 	i1 :	INT;
// 	p1 : INT;
// 	p2 : INT;
// 	p3 : INT;
// END_VAR
//
// CASE state OF
//
// 00:
// 	IF ACTIVATE AND NOT activate_last THEN
// 		state := 20;
// 		DONE := FALSE;
// 		ERROR_C := DWORD#0;
// 		ERROR_T := BYTE#0;
// 	END_IF;
//
// 20: (* URL for DNS AND HTTP-GET *)
// 	URL_DATA := STRING_TO_URL(STR:='checkip.dyndns.com',DEFAULT_PROTOCOL:='',DEFAULT_PATH:='');
// 	state := 40;
//
// 40:
// 	IF DNS_CLIENT.DONE THEN
// 		state := 60;
// 	ELSIF (DNS_CLIENT.ERROR > DWORD#00) THEN
// 		(* error handling *)
// 		ERROR_C := DNS_CLIENT.ERROR;
// 		ERROR_T := BYTE#01;
// 		state := 100;
// 	END_IF;
//
// 60:
// 	IF HTTP_GET.DONE THEN
// 		state := 80;
// 	ELSIF (HTTP_GET.ERROR > DWORD#00) THEN
// 		(* error handling *)
// 		ERROR_C := HTTP_GET.ERROR;
// 		ERROR_T := BYTE#02;
// 		state := 100;
// 	END_IF;
//
// 80:
// 	(* the following HTML page is received as the response; the IP address must be copied out of it *)
// 	(* <html><head><title>Current IP Check</title></head><body>Current IP Address: 85.127.217.33</body></html> *)
// 	st_ip := '';
// 	p1 := 0;
// 	FOR i1 := UINT_TO_INT(HTTP_GET.BODY_START) TO UINT_TO_INT(HTTP_GET.BODY_STOP) DO
// 		IF R_BUF.BUFFER[i1] = BYTE#58 THEN (* search ':' *)
// 			p1 := i1 + 2;
// 			EXIT;
// 		END_IF;
// 	END_FOR;
//
// 	p3 := p1 + 15;
// 	IF p1 > 0 AND p3 < UINT_TO_INT(HTTP_GET.BODY_STOP) THEN
// 		FOR p2 := p1 TO p3 DO
// 			IF R_BUF.BUFFER[p2] <> BYTE#60 THEN (* search '<' *)
// 				st_ip := CONCAT(st_ip,CHR_TO_STRING(C:=R_BUF.BUFFER[p2]));
// 			ELSE
// 				EXIT;
// 			END_IF;
// 		END_FOR;
// 	END_IF;
//
// 	WAN_IP4 := IP4_DECODE(STR:=st_ip);
//
// 	IF WAN_IP4 <> DWORD#0 THEN
// 		DONE := TRUE;
// 		NEW_IP4 := WAN_IP4 <> wan_ip4_last;
// 		wan_ip4_last := WAN_IP4;
// 	ELSE
// 		ERROR_C := DWORD#01; (* no valid IP found *)
// 		ERROR_T := BYTE#03;
// 	END_IF;
// 	state := 100;
//
// 100:
// 	(* UNLOCK HTTP DATA *)
// 	IF (NOT HTTP_GET.DONE) THEN
// 		state := 0;
// 		DONE := ERROR_T = BYTE#0;
// 	END_IF;
//
// END_CASE;
//
// (* ---------------- DNS --------------- *)
// DNS_CLIENT(	IP_C:=IP_C,
// 			S_BUF:=S_BUF,
// 			R_BUF:=R_BUF,
// 			DOMAIN:=URL_DATA.DOMAIN,
// 			IP4_DNS:=DWORD#00,
// 			ACTIVATE:=state=40 (* DNS Start *)
// 			);
// (* parameters not used, or not used directly *)
// (* DWORD :=DNS_CLIENT.IP4;
//    BOOL  :=DNS_CLIENT.DONE;
//    BYTE  :=DNS_CLIENT.ERROR; *)
// (* -------------------------------------*)
//
// (* ------------- HTTP_GET --------------- *)
//
// HTTP_GET(	IP_C:=IP_C,
// 			S_BUF:=S_BUF,
// 			R_BUF:=R_BUF,
// 			IP4:=DNS_CLIENT.IP4,
// 			GET:=state=60,
// 			MODE:=BYTE#2, (* HTTP 1.1 with persistent connection *)
// 			UNLOCK_BUF:=state=100,
// 			URL_DATA:=URL_DATA
// 			);
//
// (* parameters not used, or not used directly *)
// (*STRING := HTTP_GET.HTTP_STATUS;
//   UINT :=HTTP_GET.HEADER_START;
//   UINT :=HTTP_GET.HEADER_STOP;
//   UINT :=HTTP_GET.BODY_START;
//   UINT :=HTTP_GET.BODY_STOP;
//   BOOL :=HTTP_GET.DONE;
//   BYTE :=HTTP_GET.ERROR;
// *)
// (* -------------------------------------*)
//
// activate_last := ACTIVATE;
// END_FUNCTION_BLOCK

// Commented out for beedance: it uses CHR_TO_STRING, which is commented out.
// FUNCTION HTML_DECODE : STRING(STRING_LENGTH)
// VAR_INPUT
// 	IN : STRING(STRING_LENGTH);
// END_VAR
// VAR
// 	pos : INT;
// 	end : INT;
// 	tmp : STRING(10);
// 	code : STRING(1);
// END_VAR
//
// HTML_DECODE := IN;
//
// (* docode characters encoded by character position *)
// pos := FIND(HTML_DECODE, '&');
// WHILE pos > 0 DO
// 	tmp := MID(HTML_DECODE, 2, pos + 1);
// 	IF tmp = '#x' OR tmp = '#X' THEN
// 		(* hexadecimal representation found *)
// 		tmp := MID(HTML_DECODE, 10, pos + 3);
// 		end := FIND(tmp, ';');
// 		CODE := CHR_TO_STRING(DWORD_TO_BYTE(HEX_TO_DWORD(LEFT(tmp, end - 1))));
// 		HTML_DECODE := REPLACE(HTML_DECODE, CODE, end + 3, pos);
// 	ELSIF LEFT(tmp,1) = '#' THEN
// 		tmp := MID(HTML_DECODE, 10, pos + 2);
// 		end := FIND(tmp, ';');
// 		CODE := CHR_TO_STRING(INT_TO_BYTE(STRING_TO_INT(LEFT(tmp, end - 1))));
// 		HTML_DECODE := REPLACE(HTML_DECODE, CODE, end + 2, pos);
// 	ELSE
// 		(* replace all named characters *)
// 		tmp := MID(HTML_DECODE, 10, pos + 1);
// 		end := FIND(tmp, ';');
// 		CODE := CHR_TO_STRING(CHARCODE(LEFT(tmp, end - 1)));
// 		HTML_DECODE := REPLACE(HTML_DECODE, CODE, end + 1, pos);
// 	END_IF;
// 	(* search for next occurence of encoded characters *)
// 	pos := FINDP(HTML_DECODE, '&', pos + 1);
// END_WHILE;
// END_FUNCTION

// Commented out for beedance: it reads or writes the bytes of a STRING through a pointer; a beedance reference (REF_TO) refers to a whole variable of its type.
// FUNCTION HTML_ENCODE : STRING(STRING_LENGTH)
// VAR_INPUT
// 	IN : STRING(STRING_LENGTH);
// 	M : BOOL;
// END_VAR
// VAR
// 	pt_in : REF_TO ARRAY[1..255] OF BYTE;
// 	pt_out : REF_TO ARRAY[1..256] OF BYTE;
// 	pos_in : INT;
// 	pos_out : INT;
// 	stop : INT;
// 	B: BYTE;
// 	tmp : STRING(10);
// 	i: INT;
// END_VAR
//
// pt_in  := REF(in);
// pt_out := REF(HTML_ENCODE);
//
// (* scan the input string and convert unallowed characters *)
// pos_in := 1;
// stop := LEN(in);
// FOR pos_out := 1 TO 250 DO
// 	IF pos_in > stop THEN EXIT; END_IF;
// 	B := pt_in^[pos_in];
// 	CASE BYTE_TO_INT(B) OF
// 		34: (* " detected *)
// 			IF pos_out > STRING_LENGTH - 6 THEN EXIT; END_IF;
// 			pt_out^[pos_out] := 38;
// 			pos_out := pos_out + 1;
// 			pt_out^[pos_out] := 113;
// 			pos_out := pos_out + 1;
// 			pt_out^[pos_out] := 117;
// 			pos_out := pos_out + 1;
// 			pt_out^[pos_out] := 111;
// 			pos_out := pos_out + 1;
// 			pt_out^[pos_out] := 116;
// 			pos_out := pos_out + 1;
// 			pt_out^[pos_out] := 59;
// 		38: (* & detected *)
// 			IF pos_out > STRING_LENGTH - 5 THEN EXIT; END_IF;
// 			pt_out^[pos_out] := 38;
// 			pos_out := pos_out + 1;
// 			pt_out^[pos_out] := 97;
// 			pos_out := pos_out + 1;
// 			pt_out^[pos_out] := 109;
// 			pos_out := pos_out + 1;
// 			pt_out^[pos_out] := 112;
// 			pos_out := pos_out + 1;
// 			pt_out^[pos_out] := 59;
// 		60: (* < detected *)
// 			IF pos_out > STRING_LENGTH - 4 THEN EXIT; END_IF;
// 			pt_out^[pos_out] := 38;
// 			pos_out := pos_out + 1;
// 			pt_out^[pos_out] := 108;
// 			pos_out := pos_out + 1;
// 			pt_out^[pos_out] := 116;
// 			pos_out := pos_out + 1;
// 			pt_out^[pos_out] := 59;
// 		62: (* > detected *)
// 			IF pos_out > STRING_LENGTH - 4 THEN EXIT; END_IF;
// 			pt_out^[pos_out] := 38;
// 			pos_out := pos_out + 1;
// 			pt_out^[pos_out] := 103;
// 			pos_out := pos_out + 1;
// 			pt_out^[pos_out] := 116;
// 			pos_out := pos_out + 1;
// 			pt_out^[pos_out] := 59;
// 	ELSE
// 		IF M AND B > 127 THEN
// 			tmp := CHARNAME(B);
// 			(* exit if output string has not enough space *)
// 			IF pos_out + LEN(tmp) + 2 <= 250 THEN
// 				pt_out^[pos_out] := 38;
// 				pos_out := pos_out + 1;
// 				FOR i := 1 TO LEN(tmp) DO
// 					pt_out^[pos_out] := CODE(tmp, i);
// 					pos_out := pos_out + 1;
// 				END_FOR;
// 				pt_out^[pos_out] := 59;
// 			END_IF;
// 		ELSE
// 			pt_out^[pos_out] := B;
// 		END_IF;
// 	END_CASE;
// 	(* increment in by 1 *)
// 	pos_in := pos_in + 1;
// END_FOR;
//
// (* terminate the output string *)
// pt_out^[pos_out] := 0;
// END_FUNCTION

// Commented out for beedance: it uses _STRING_TO_BUFFER, which is commented out.
// FUNCTION_BLOCK HTTP_GET
// VAR_IN_OUT
// 	URL_DATA : url;
// 	IP_C : IP_C; (* IP_Control management structure *)
// 	S_BUF : NETWORK_BUFFER;
// 	R_BUF : NETWORK_BUFFER;
// END_VAR
// VAR_INPUT
// 	IP4 : DWORD;
// 	GET : BOOL;
// 	MODE : BYTE := BYTE#2;
// 	UNLOCK_BUF : BOOL;
// END_VAR
// VAR_OUTPUT
// 	HTTP_STATUS : STRING;
// 	HEADER_START : UINT; (* HTTP Header (Message Header) *)
// 	HEADER_STOP : UINT; (* HTTP Header (Message Header) *)
// 	BODY_START : UINT; (* Message Body *)
// 	BODY_STOP : UINT; (* Message Body *)
// 	DONE : BOOL;
// 	ERROR : DWORD;
// END_VAR
// VAR
// 	READ_HTTP :	READ_HTTP;
// 	BASE64_ENCODE_STR :	BASE64_ENCODE_STR;
// 	b64_str1 :	STRING(144);
// 	b64_str2 :	STRING(192);
// 	b64_done :	BOOL;
// 	b64_start :	BOOL;
// 	authentication :	BOOL;
// 	IP_FIFO : IP_FIFO;
// 	ip_state : BYTE;
// 	ip_id : BYTE;
// 	get_last : BOOL;
// 	ip4_stored : DWORD;
// 	state : INT;
// 	i : INT;
// 	http_1_1_host : BOOL;
// 	total_size : INT;
// 	text : STRING(STRING_LENGTH);
// 	delimiter2b : STRING(2);
// 	delimiter4b : STRING(4);
// 	del_end : STRING(4);
// 	del_pos : INT;
// 	idx : INT;
// 	rcv_timeout : BOOL;
// 	con_rdce : BOOL;
//
// 	(*LOG_MSG : LOG_MSG;
// 	_debug_enable : BOOL := TRUE;
// 	_debug_state_last : INT := -1;*)
//
// END_VAR
//
// CASE state OF
// 00:	DONE := FALSE;
// 	IF GET AND NOT GET_LAST THEN (* wait for rising edge on SET *)
// 		state := 10;
// 		ip4_stored := IP4; (* store current IP4 *)
// 		total_size := 0;
// 		HEADER_START := UINT#0;
// 		HEADER_STOP := UINT#0;
// 		BODY_START := UINT#0;
// 		BODY_STOP := UINT#0;
// 		HTTP_STATUS := '';
// 		ERROR := DWORD#0;
// 		ip_state := BYTE#1; (* register *)
// 		authentication := FALSE;
// 		delimiter2b := '$0D$0A';
// 		delimiter4b := '$0D$0A$0D$0A';
//
// 		(* LOGIN parameters present *)
// 		(* LOGIN parameters present *)
// 		IF URL_DATA.USER <> '' AND URL_DATA.PASSWORD <> '' THEN
// 			b64_str1 := CONCAT(URL_DATA.USER,':');
// 			b64_str1 := CONCAT(b64_str1,URL_DATA.PASSWORD); (* USER:PASSWORD *)
// 			b64_start := TRUE; (* BASE64 encoding of username *)
// 			authentication := TRUE;
// 			state := 5;
// 		ELSE
// 			state := 10;
// 		END_IF;
// 	        	(*####################  DEBUG-MESSAGE  ###################################*)
// 		(*IF _debug_enable THEN
// 	       		LOG_CL.NEW_MSG := 'HTTP: S00 START /IP_ID ~4';
// 	            	LOG_CL.PRINTF[4]  := BYTE_TO_STRING(IP_ID);
// 	            	LOG_MSG();
// 	        	END_IF;*)
// 	        	(*########################################################################*)
// 	END_IF;
//
// 5:	IF b64_start AND b64_done THEN (* wait for base64 conversion *)
// 		b64_start := FALSE;
// 		state := 10;
// 	END_IF;
//
// 10:	IF ip_state = BYTE#3 THEN (* register with IP_Control and wait for release *)
// 		idx := 0;
// 		text := CONCAT('GET ',URL_DATA.PATH);
// 		_STRING_TO_BUFFER(STR:=text,POS:=idx,PT:=REF(S_BUF.BUFFER),SIZE:=SIZEOF(S_BUF.BUFFER)); (* copy GET path into buffer *)
// 		idx := idx + LEN(text);
//
// 		IF LEN(URL_DATA.QUERY) > 0 THEN
// 			S_BUF.BUFFER[idx] := 63; (* ASCII '?' *)
// 			idx := idx + 1;
// 			_STRING_TO_BUFFER(STR:=URL_DATA.QUERY,POS:=idx,PT:=REF(S_BUF.BUFFER),SIZE:=SIZEOF(S_BUF.BUFFER)); (* copy QUERY into buffer *)
// 			idx := idx + LEN(URL_DATA.QUERY);
// 		END_IF;
//
// 		IF MODE >= BYTE#2 THEN (* pass requested HTTP version *)
// 			text := ' HTTP/1.1';
// 		ELSE
// 			text := ' HTTP/1.0';
// 		END_IF;
// 		text := CONCAT(text,delimiter2b);
// 		_STRING_TO_BUFFER(STR:=text,POS:=idx,PT:=REF(S_BUF.BUFFER),SIZE:=SIZEOF(S_BUF.BUFFER)); (* copy HTTP version into buffer *)
// 		idx := idx + LEN(text);
//
// 		IF MODE = BYTE#1 THEN (* HTTP/1.0 with persistent connection requested *)
// 			text := CONCAT('Connection: Keep-Alive',delimiter2b); (* workaround for pcworx -> $0D$0A not possible as a string constant *)
// 		ELSIF MODE = BYTE#3 THEN (* HTTP/1.1 without persistent connection requested *)
// 			text := CONCAT('Connection: Close',delimiter2b); (* workaround for pcworx -> $0D$0A not possible as a string constant *)
// 		ELSE
// 			text := '';
// 		END_IF;
//
// 		(* take additional parameters *)
// 		text := CONCAT(text,URL_DATA.HEADER);
// 		_STRING_TO_BUFFER(STR:=text,POS:=idx,PT:=REF(S_BUF.BUFFER),SIZE:=SIZEOF(S_BUF.BUFFER)); (* copy HTTP version into buffer *)
// 		idx := idx + LEN(text);
//
// 		IF authentication THEN
// 			text := CONCAT('Authorization: Basic ',b64_str2);
// 			text := CONCAT(text,delimiter2b); (* workaround for pcworx -> $0D$0A not possible as a string constant *)
// 			_STRING_TO_BUFFER(STR:=text,POS:=idx,PT:=REF(S_BUF.BUFFER),SIZE:=SIZEOF(S_BUF.BUFFER)); (* copy HTTP host into buffer *)
// 			idx := idx + LEN(text);
// 		END_IF;
//
// 		text := CONCAT('Host: ',URL_DATA.DOMAIN);
// 		text := CONCAT(text,delimiter4b); (* workaround for pcworx -> $0D$0A not possible as a string constant *)
// 		_STRING_TO_BUFFER(STR:=text,POS:=idx,PT:=REF(S_BUF.BUFFER),SIZE:=SIZEOF(S_BUF.BUFFER)); (* copy HTTP host into buffer *)
// 		idx := idx + LEN(text);
//
// 		(* set up IP data traffic *)
// 		IF FIND(';HTTPS;https;Https;', CONCAT(URL_DATA.PROTOCOL,';')) > 1 THEN
// 			IP_C.C_PORT := SEL(URL_DATA.PORT = WORD#0,URL_DATA.PORT,WORD#443); (* enter port number *)
// 			IP_C.MAILBOX[16] := BYTE#1; (* enable SSL mode *)
// 		ELSE
// 			IP_C.C_PORT := SEL(URL_DATA.PORT = WORD#0,URL_DATA.PORT,WORD#80);  (* enter port number *)
// 		END_IF;
//
// 		IP_C.C_IP := ip4_stored; (* enter IP *)
// 		IP_C.C_MODE := BYTE#0; (* Mode: TCP+ACTIVE+PORT+IP *)
// 		IP_C.C_ENABLE := TRUE; (* enable connection setup *)
// 		IP_C.TIME_RESET := TRUE; (* reset timeout monitoring *)
// 		IP_C.R_OBSERVE := TRUE; (* monitor data reception *)
// 		S_BUF.SIZE := INT_TO_UINT(idx); (* enter send length *)
// 		R_BUF.SIZE := UINT#0; (* reset receive length *)
//
// 		state := 30;
// 	        	(*####################  DEBUG-MESSAGE  ###################################*)
// 	        	(*IF _debug_enable THEN
// 	        		LOG_CL.NEW_MSG := 'HTTP: S20 SEND /IP_ID ~4';
// 	            	LOG_CL.PRINTF[4]  := BYTE_TO_STRING(IP_ID);
// 	            	LOG_MSG();
// 	        	END_IF;*)
// 	        	(*########################################################################*)
// 	END_IF;
//
// 30:	rcv_timeout := (IP_C.ERROR AND DWORD#16#0000_FF00) = DWORD#16#0000_FF00;
// 	con_rdce :=     (IP_C.ERROR AND DWORD#16#FD00_0000) = DWORD#16#FD00_0000;
//
// 	IF S_BUF.SIZE = UINT#0 THEN
// 		IF total_size = 0 THEN
// 			IF R_BUF.SIZE > UINT#15 THEN; (* check length of received data *)
//
// 				(* search end of HTTP HEADER -> recognizable by $0D$A$0D$A on DEC RT-11,CP/M,MS-DOS,Windows *)
// 				del_end := '$0D$0A$0D$0A';
// 				del_pos := BUFFER_SEARCH(PT:=REF(R_BUF.BUFFER),SIZE:=R_BUF.SIZE,STR:=del_end,POS:=0,IGN:=FALSE);
//
// 				(* no end found? -> search other end encoding *)
// 				IF del_pos = 0 THEN
// 					del_end := '$0A$0A';
// 					(* search end of HTTP HEADER -> recognizable by $0A$0A on Multics, Unix derivatives, Mac OS X *)
// 					del_pos := BUFFER_SEARCH(PT:=REF(R_BUF.BUFFER),SIZE:=R_BUF.SIZE,STR:=del_end,POS:=0,IGN:=FALSE);
// 				END_IF;
//
// 				IF del_pos > 0 THEN
// 					HEADER_START := UINT#0;
// 					HEADER_STOP := INT_TO_UINT(del_pos + LEN(del_end) - 1);
// 					TOTAL_SIZE := -1; (* HTTP header received but total length not known yet *)
// 				END_IF;
// 		                	(*####################  DEBUG-MESSAGE  ###################################*)
// 		                	(*IF _debug_enable THEN
// 		                   	LOG_CL.NEW_MSG := 'HTTP: S20 HEADER_START ~1 / HEADER_STOP ~2/IP_ID ~4';
// 		                   	LOG_CL.PRINTF[4]  := BYTE_TO_STRING(IP_ID);
// 		                   	LOG_CL.PRINTF[1]  := UINT_TO_STRING(HEADER_START);
// 		                   	LOG_CL.PRINTF[2]  := UINT_TO_STRING(HEADER_STOP);
// 		                   	LOG_MSG();
// 		                	END_IF;*)
// 		                	(*########################################################################*)
//
// 				(* evaluate HTTP status code: (can be 1.0 or 1.1 *)
// 				READ_HTTP(size:=HEADER_STOP,pos:=0,SRC:='',pt:=R_BUF.BUFFER);
//
// 				i := LEN(READ_HTTP.READ_HTTP);
// 				IF i > 7 THEN
// 					(* evaluate HTTP version of HOST 1.0 or 1.1 *)
// 					text:=MID(READ_HTTP.READ_HTTP,1,3);
// 					http_1_1_host := text = '1';
//
// 					(* isolate code and message *)
// 					HTTP_STATUS := RIGHT(READ_HTTP.READ_HTTP,i-4);
// 				END_IF;
//
// 				(* positive HTTP request? *)
// 				IF FIND(HTTP_STATUS,'200') > 0 THEN
//
// 					(* 'Content-Length: read and evaluate value *)
// 					READ_HTTP(size:=HEADER_STOP,pos:=0,SRC:='CONTENT-LENGTH',pt:=R_BUF.BUFFER);
// 					text:=READ_HTTP.READ_HTTP;
//
// 					IF LEN(text) >= 1 THEN
// 						IF IS_NUM(str:=text) THEN
// 							(* calculate expected total number of bytes *)
// 							total_size := STRING_TO_INT(text) + UINT_TO_INT(HEADER_STOP) + 1;
//                            					(*####################  DEBUG-MESSAGE  ###################################*)
//                            					(*IF _debug_enable THEN
//                               					LOG_CL.NEW_MSG := 'HTTP: S20 HEADER ~1, BODY ~2 TOTAL ~3 /IP_ID ~4';
//                              					LOG_CL.PRINTF[4]  := BYTE_TO_STRING(IP_ID);
//                                					LOG_CL.PRINTF[1]  := UINT_TO_STRING(HEADER_STOP);
//                                					LOG_CL.PRINTF[2]  := INT_TO_STRING(TOTAL_SIZE-UINT_TO_INT(HEADER_STOP));
//                                					LOG_CL.PRINTF[3]  := INT_TO_STRING(TOTAL_SIZE);
//                               					LOG_MSG();
//                           					END_IF;*)
//                           					(*########################################################################*)
// 						END_IF;
// 					END_IF;
// 				ELSE
// 					ERROR := DWORD#16#000000FC; (* error from HTTP status codes *)
// 				END_IF;
// 			END_IF;
// 		(* 1. with a known Content-Length the connection is closed after the expected data is received *)
// 		(* 2. with a persistent connection and unknown data amount, wait for the receive timeout *)
// 		(* 3. if the host closes the connection after data was received *)
// 		ELSIF (R_BUF.SIZE >= INT_TO_UINT(total_size)) OR
// 			(R_BUF.SIZE > UINT#0 AND total_size < 0 AND ((rcv_timeout OR con_rdce) OR (IP_C.C_STATE = BYTE#1))) THEN
//
// 			IF R_BUF.SIZE - 1 > HEADER_STOP THEN (* BODY data present *)
// 				BODY_START := HEADER_STOP + UINT#1;
// 				BODY_STOP := R_BUF.SIZE - 1;
// 		                	(*####################  DEBUG-MESSAGE  ###################################*)
// 		                	(*IF _debug_enable THEN
// 		                   	LOG_CL.NEW_MSG := 'HTTP: S20 BODY ~1, START ~2 END ~3 /IP_ID ~4';
// 		                   	LOG_CL.PRINTF[4]  := BYTE_TO_STRING(IP_ID);
// 		                   	LOG_CL.PRINTF[1]  := UINT_TO_STRING(HEADER_STOP);
// 		                   	LOG_CL.PRINTF[2]  := UINT_TO_STRING(BODY_START);
// 		                   	LOG_CL.PRINTF[3]  := UINT_TO_STRING(BODY_STOP);
// 		                   	LOG_MSG();
// 		               	END_IF;*)
// 		               	(*########################################################################*)
// 			END_IF;
//
// 			DONE := TRUE;
// 			IP_C.C_ENABLE := FALSE; (* close connection *)
// 			state := 40;
//             		(*####################  DEBUG-MESSAGE  ###################################*)
//             		(*IF _debug_enable THEN
//                 			LOG_CL.NEW_MSG := 'HTTP: S30 OK /IP_ID ~4';
//                 			LOG_CL.PRINTF[4]  := BYTE_TO_STRING(IP_ID);
//                 			LOG_MSG();
//             		END_IF;*)
//             		(*########################################################################*)
// 		END_IF;
// 	END_IF;
//
// 	IF IP_C.ERROR <> DWORD#0 THEN
// 		(* with unknown content size it is not known whether or how many telegrams will still follow *)
// 		(* so after a receive timeout or remote disconnect error the error is filtered out again (logical error) *)
// 		IF rcv_timeout AND DONE THEN
// 			IP_C.ERROR := IP_C.ERROR AND DWORD#16#FFFF_00FF; (* reset error again *)
// 		ELSIF con_rdce AND DONE THEN
// 			IP_C.ERROR := IP_C.ERROR AND DWORD#16#00FF_FFFF; (* reset error again *)
// 		ELSE
// 			ERROR := IP_C.ERROR;
// 		END_IF;
// 	END_IF;
//
// 	IF ERROR > DWORD#0 THEN
// 		IP_C.C_ENABLE := FALSE; (* block connection setup *)
// 		state := 40;
// 	        	(*####################  DEBUG-MESSAGE  ###################################*)
// 	        	(*IF _debug_enable THEN
// 	            	LOG_CL.NEW_MSG := 'HTTP: S30 ERROR ~1 /IP_ID ~4';
// 	            	LOG_CL.PRINTF[1]  := DWORD_TO_STRING(ERROR);
// 	            	LOG_CL.PRINTF[4]  := BYTE_TO_STRING(IP_ID);
// 	            	LOG_MSG();
// 	        	END_IF;*)
// 	        	(*########################################################################*)
// 	END_IF;
//
// 40:	IF (UNLOCK_BUF OR NOT DONE) THEN (* wait for release and connection closed -> remove IP_ID from stack *)
// 		IP_STATE := BYTE#4; (* unregister *)
// 		DONE := FALSE;
// 		IP_C.MAILBOX[16] := BYTE#0; (* end SSL mode *)
// 		state := 0;
// 	END_IF;
// END_CASE;
//
// get_last := GET; (* save last status for edge detection *)
//
// IP_FIFO(FIFO:=IP_C.FIFO,STATE:=ip_state,ID:=ip_id); (* IP_FIFO *)
//
// BASE64_ENCODE_STR(RUN:=b64_start,STR1:=b64_str1,STR2:=b64_str2); (* BASE64 encoding *)
// b64_done:=BASE64_ENCODE_STR.DONE;
//
// (*####################  DEBUG-MESSAGE  ###################################*)
// (*IF _debug_enable THEN
// 	IF state <> _debug_state_last THEN
// 		LOG_CL.NEW_MSG := 'http_get: /last ~1 /New ~2';
// 		LOG_CL.PRINTF[1] := INT_TO_STRING(_debug_state_last);
// 		LOG_CL.PRINTF[2] := INT_TO_STRING(state);
// 		LOG_MSG();
// 		_debug_state_last := state;
// 	END_IF;
// END_IF;*)
// (*########################################################################*)
// END_FUNCTION_BLOCK

// Commented out for beedance: it reads or writes the bytes of a STRING through a pointer; a beedance reference (REF_TO) refers to a whole variable of its type.
// FUNCTION_BLOCK INI_PARSER_BUF
// VAR_IN_OUT
// 	STR : STRING(STRING_LENGTH);
// 	RUN : BYTE;
// 	OFFSET : UDINT;
// 	KEY : STRING(STRING_LENGTH);
// 	VALUE : STRING(STRING_LENGTH);
// 	PT : NETWORK_BUFFER;
// END_VAR
// VAR_OUTPUT
// 	RESULT : BYTE;
// END_VAR
// VAR
// 	step : INT;
// 	size : INT;
// 	c : BYTE;
// 	k_add : BYTE;
// 	v_add : BYTE;
// 	i : INT;
// 	state : BYTE;
// 	eof : BOOL;
// 	pv : REF_TO BYTE;
// 	pk : REF_TO BYTE;
// 	pve : DWORD;
// 	pke : DWORD;
// 	watchdog : TON;
//
// 	(*LOG_MSG : LOG_MSG;
// 	_debug_enable : BOOL := TRUE;
// 	step_last : INT;*)
// END_VAR
//
// IF RUN > 0 THEN
// 	IF state = 0 THEN (* restart evaluation *)
//
// 		pv := REF(VALUE);
// 		pv^ := 0; (* VALUE = '' *)
// 		pve := pv + INT_TO_DWORD(STRING_LENGTH);
// 		pk := REF(KEY);
// 		pk^ := 0; (* KEY = '' *)
// 		pke := pk + INT_TO_DWORD(STRING_LENGTH);
//
// 		i := UDINT_TO_INT(OFFSET);
// 		size := UINT_TO_INT(PT.SIZE) - 1;
// 		RESULT := 0;
// 		state := 5; (* command in progress (busy) *)
// 		step := 0; (* restart evaluation *)
//
// 		(*####################  DEBUG-MESSAGE  ###################################*)
// 		(*IF _debug_enable THEN
// 			LOG_CL.NEW_MSG := 'IPB: Startindex: ~1';
// 			LOG_CL.PRINTF[1]  := INT_TO_STRING(i);
// 			LOG_MSG();
// 		END_IF;*)
// 		(*########################################################################*)
// 	END_IF;
//
// 	watchdog(IN:=FALSE,PT:=T#1ms); (* restart timer *)
// 	watchdog.IN := TRUE;
//
// 	WHILE (state = 5) DO (* loop as long as there is no result *)
//
// 		watchdog(); (* update timer *)
//
// 		IF watchdog.Q THEN (* watchdog triggered *)
// 			state := 5;
// 			EXIT;
// 		ELSIF i > size THEN (* no further character available *)
// 			state := 10; (* nothing found - end of data reached *)
// 			EXIT;
// 		ELSE
//
// 			c := PT.BUFFER[i]; (* read new character from buffer *)
// 			eof := i + 1 = PT.SIZE; (* End of File *)
//
// 			k_add := 0;
// 			v_add := 0;
//
// 			CASE step OF
//
// 			0: (* no mode detected yet *)
// 				IF c = 91 THEN (* compare with "[" *)
// 					step := 200; (* activate mode for section *)
// 				ELSIF c = 59 OR c = 35 THEN (* compare with ";" and '#' *)
// 					step := 100; (* activate mode for comment *)
// 				ELSIF c > 32 THEN (* key detected *)
// 					k_add := c; (* store character *)
// 					step := 300; (* start key evaluation *)
// 				END_IF;
// 			100: (* comment detected -> search end of line *)
// 				IF c < 32 THEN (* check for control characters *)
// 					state  := 3; (* exit -> comment was found *)
// 				END_IF;
// 			200: (* section start detected -> search section end *)
// 				IF c = 93 THEN (* compare with "]" *)
// 					IF pk > REF(KEY) > 0 THEN (* there must be at least one character inside [] *)
// 						state  := 1; (* exit -> section was found *)
// 					ELSE
// 						pk := REF(KEY);
// 						pk^ := 0; (* KEY = '' *)
// 						step := 0; (* faulty section line present -> continue searching *)
// 					END_IF;
// 				ELSIF c < 32 OR eof THEN (* control character - faulty section line -> continue searching *)
// 					pk := REF(KEY);
// 					pk^ := 0; (* KEY = '' *)
// 					step := 0;
// 				ELSE
// 					k_add := c; (* store character *)
// 				END_IF;
// 			300: (* begin: key detected -> evaluate name *)
// 				IF c < 32 THEN (* control character - faulty key line -> continue searching *)
// 					pk := REF(KEY);
// 					pk^ := 0; (* KEY = '' *)
// 					step := 0;
// 				ELSIF c = 61 THEN (* check for '=' *)
// 					step := 330;
// 				ELSE
// 					k_add := c; (* store character *)
// 				END_IF;
// 			330: (* search KeyValue start *)
// 				IF c < 32 THEN (* control character  *)
// 					state := 2; (* key without value found *)
// 				ELSIF eof THEN
// 					state := 2; (* key without value found *)
// 					v_add := c; (* store character *)
// 				ELSE
// 					v_add := c; (* store character *)
// 					step := 350;
// 				END_IF;
// 			350: (* search KeyValue end *)
// 				IF c < 32 THEN (* control character *)
// 					state := 2; (* key found *)
// 				ELSIF eof THEN
// 					v_add := c; (* store character *)
// 					state := 2; (* key found *)
// 				ELSE
// 					v_add := c; (* store character *)
// 				END_IF;
// 			END_CASE;
//
// 			IF v_add > 0  AND pv < pve THEN (* add character to value string *)
// 				pv^ := v_add; (* enter character *)
// 				pv := pv + 1;
// 				pv^ := 0; (* enter string termination *)
// 			END_IF;
//
// 			IF k_add > 0 AND pk < pke THEN (* add character to key string *)
// 				pk^ := k_add; (* enter character *)
// 				pk := pk + 1;
// 				pk^ := 0; (* enter string termination *)
// 			END_IF;
//
// 			i := i + 1; (* increment data pointer *)
//
// 		END_IF;
// 	END_WHILE;
//
// 	CASE state OF
// 	01:	(* section found *)
// 		IF RUN = 1 OR RUN = 3 THEN (* section preselected or report everything *)
// 			IF KEY = STR OR LEN(STR) = 0 THEN (* compare with searched section or no section specified *)
// 				RESULT := 1; (* section found *)
// 				OFFSET := i; (* take offset *)
// 				RUN := 0;
// 				state := 0;
// 			END_IF;
// 		ELSE
// 			pk := REF(KEY);
// 			pk^ := 0; (* KEY = '' *)
// 			RESULT := 11; (* key not found, section end - do not change offset *)
// 			RUN := 0;
// 			state := 0;
// 		END_IF;
// 	02:	(* key found *)
// 		IF RUN = 2 OR RUN = 3 THEN (* key preselected or report everything *)
// 			IF KEY = STR OR LEN(STR) = 0 THEN (* compare with searched key *)
// 				RESULT := 2; (* key found *)
// 				OFFSET := i; (* take offset *)
// 				RUN := 0;
// 				state := 0;
// 			END_IF;
// 		END_IF;
// 	03:	(* comment found *)
// 		OFFSET := i; (* take offset *)
// 		state := 0;
//
// 	05:	RESULT := 5; (* in progress *)
//
// 	10:	(* index out of range - end of buffer *)
// 		RESULT := 10; (* nothing found - end of data reached *)
// 		OFFSET := i; (* take offset *)
// 		RUN := 0;
// 		state := 0;
// 	END_CASE;
//
// 	(*####################  DEBUG-MESSAGE  ###################################*)
// 	(*IF _debug_enable THEN
// 		LOG_CL.NEW_MSG := 'IPF: intern Result ~1 , state ~2, step ~3 , offset ~4, run ~5';
// 		LOG_CL.PRINTF[1] := BYTE_TO_STRING(RESULT);
// 		LOG_CL.PRINTF[2] := BYTE_TO_STRING(state);
// 		LOG_CL.PRINTF[3] := INT_TO_STRING(step);
// 		LOG_CL.PRINTF[4] := UDINT_TO_STRING(OFFSET);
// 		LOG_CL.PRINTF[5] := BYTE_TO_STRING(RUN);
// 		LOG_MSG();
// 	END_IF;*)
// 	(*########################################################################*)
//
// END_IF;
//
// (*####################  DEBUG-MESSAGE  ###################################*)
// (*IF _debug_enable THEN
// 	IF step_last <> step THEN
// 		LOG_CL.NEW_MSG := 'IPB: Step: ~1';
// 		LOG_CL.PRINTF[1]  := INT_TO_STRING(step);
// 		LOG_MSG();
// 	END_IF;
// 	step_last := step;
// END_IF;*)
// (*########################################################################*)
// END_FUNCTION_BLOCK

// Commented out for beedance: it reads or writes the bytes of a STRING through a pointer; a beedance reference (REF_TO) refers to a whole variable of its type.
// FUNCTION_BLOCK INI_PARSER_FILE
// VAR_IN_OUT
// 	FILENAME : STRING;
// 	FSD : FILE_SERVER_DATA	;
// 	STR : STRING(STRING_LENGTH);
// 	RUN : BYTE;
// 	OFFSET : UDINT;
// 	KEY : STRING(STRING_LENGTH);
// 	VALUE : STRING(STRING_LENGTH);
// 	PT	: NETWORK_BUFFER;
// END_VAR
// VAR_OUTPUT
// 	RESULT : BYTE;
// END_VAR
// VAR
// 	FB : FILE_BLOCK;
// 	i : UDINT;
// 	state : BYTE;
// 	e : BYTE;
// 	mode : BYTE;
// 	step : INT;
// 	c : BYTE;
// 	k_add : BYTE;
// 	v_add : BYTE;
// 	eof : BOOL;
// 	pv : REF_TO BYTE;
// 	pk : REF_TO BYTE;
// 	pve : DWORD;
// 	pke : DWORD;
// 	watchdog : TON;
//
// 	(*LOG_MSG : LOG_MSG;
// 	_debug_enable : BOOL := TRUE;
// 	step_last : INT;*)
// END_VAR
//
// IF RUN > 0 THEN
//
// 	IF state = 0 THEN (* restart evaluation *)
// 		pv := REF(VALUE);
// 		pv^ := 0; (* VALUE = '' *)
// 		pve := pv + INT_TO_DWORD(STRING_LENGTH);
// 		pk := REF(KEY);
// 		pk^ := 0; (* KEY = '' *)
// 		pke := pk + INT_TO_DWORD(STRING_LENGTH);
//
// 		i := OFFSET;
// 		RESULT := 0;
// 		state := 5; (* command in progress (busy) *)
// 		step := 0; (* restart evaluation *)
//
// 		(*####################  DEBUG-MESSAGE  ###################################*)
// 		(*IF _debug_enable THEN
// 			LOG_CL.NEW_MSG := 'IPF: Startindex: ~1';
// 			LOG_CL.PRINTF[1] := UDINT_TO_STRING(i);
// 			LOG_MSG();
// 		END_IF;*)
// 		(*########################################################################*)
//
// 	END_IF;
//
// 	watchdog(IN:=FALSE,PT:=T#1ms); (* restart timer *)
// 	watchdog.IN := TRUE;
//
// 	WHILE (state = 5) DO (* loop as long as there is no result *)
//
// 		mode := 1;
// 		FB(MODE:=mode,FSD:=fsd,PT:=PT,FILENAME:=FILENAME,POS:=i );
// 		e:=FB.ERROR;
// 		c:=FB.DATA;
//
// 		eof := i + 1 = FSD.FILE_SIZE; (* End of File *)
//
// 		(*####################  DEBUG-MESSAGE  ###################################*)
// 		(*IF _debug_enable THEN
// 			LOG_CL.NEW_MSG := 'IPF: mode: ~1, error: ~2 , >~7<>~3< ~4 step ~5 index ~6';
// 			LOG_CL.PRINTF[1] := BYTE_TO_STRING(mode);
// 			LOG_CL.PRINTF[2] := BYTE_TO_STRING(e);
// 			LOG_CL.PRINTF[3] := BYTE_TO_STRING(c);
// 			LOG_CL.PRINTF[4] := BOOL_TO_STRING(eof);
// 			LOG_CL.PRINTF[5] := INT_TO_STRING(step);
// 			LOG_CL.PRINTF[6] := UDINT_TO_STRING(i);
// 			LOG_CL.PRINTF[7] := CHR_TO_STRING(c);
// 			LOG_MSG();
// 		END_IF;*)
// 		(*########################################################################*)
//
// 		watchdog(); (* update timer *)
//
// 		IF mode > 0 OR watchdog.Q THEN (* block still active, or watchdog triggered *)
// 			state := 5;
// 			EXIT;
// 		ELSIF e > 0 THEN (* File_error or no further character available *)
// 			state := 10; (* nothing found - end of data reached *)
// 			EXIT;
// 		ELSE
//
// 			k_add := 0;
// 			v_add := 0;
//
// 			CASE step OF
//
// 			0: (* no mode detected yet *)
// 				IF c = 91 THEN (* compare with "[" *)
// 					step := 200; (* activate mode for section *)
// 				ELSIF c = 59 OR c = 35 THEN (* compare with ";" and '#' *)
// 					step := 100; (* activate mode for comment *)
// 				ELSIF c > 32 THEN (* key detected *)
// 					k_add := c; (* store character *)
// 					step := 300; (* start key evaluation *)
// 				END_IF;
// 			100: (* comment detected -> search end of line *)
// 				IF c < 32 THEN (* check for control characters *)
// 					state  := 3; (* exit -> comment was found *)
// 				END_IF;
// 			200: (* section start detected -> search section end *)
// 				IF c = 93 THEN (* compare with "]" *)
// 					IF pk > REF(KEY) > 0 THEN (* there must be at least one character inside [] *)
// 						state  := 1; (* exit -> section was found *)
// 					ELSE
// 						pk := REF(KEY);
// 						pk^ := 0; (* KEY = '' *)
// 						step := 0; (* faulty section line present -> continue searching *)
// 					END_IF;
// 				ELSIF c < 32 OR eof THEN (* control character - faulty section line -> continue searching *)
// 					pk := REF(KEY);
// 					pk^ := 0; (* KEY = '' *)
// 					step := 0;
// 				ELSE
// 					k_add := c; (* store character *)
// 				END_IF;
// 			300: (* begin: key detected -> evaluate name *)
// 				IF c < 32 THEN (* control character - faulty key line -> continue searching *)
// 					pk := REF(KEY);
// 					pk^ := 0; (* KEY = '' *)
// 					step := 0;
// 				ELSIF c = 61 THEN (* check for '=' *)
// 					step := 330;
// 				ELSE
// 					k_add := c; (* store character *)
// 				END_IF;
// 			330: (* search KeyValue start *)
// 				IF c < 32 THEN (* control character  *)
// 					state := 2; (* key without value found *)
// 				ELSIF eof THEN
// 					state := 2; (* key without value found *)
// 					v_add := c; (* store character *)
// 				ELSE
// 					v_add := c; (* store character *)
// 					step := 350;
// 				END_IF;
// 			350: (* search KeyValue end *)
// 				IF c < 32 THEN (* control character *)
// 					state := 2; (* key found *)
// 				ELSIF eof THEN
// 					v_add := c; (* store character *)
// 					state := 2; (* key found *)
// 				ELSE
// 					v_add := c; (* store character *)
// 				END_IF;
// 			END_CASE;
//
// 			IF v_add > 0  AND pv < pve THEN (* add character to value string *)
// 				pv^ := v_add; (* enter character *)
// 				pv := pv + 1;
// 				pv^ := 0; (* enter string termination *)
// 			END_IF;
//
// 			IF k_add > 0 AND pk < pke THEN (* add character to key string *)
// 				pk^ := k_add; (* enter character *)
// 				pk := pk + 1;
// 				pk^ := 0; (* enter string termination *)
// 			END_IF;
//
// 			i := i + 1; (* increment data pointer *)
//
// 		END_IF;
// 	END_WHILE;
//
// 	CASE state OF
// 	01:	(* section found *)
// 		IF RUN = 1 OR RUN = 3 THEN (* section preselected or report everything *)
// 			IF KEY = STR OR LEN(STR) = 0 THEN (* compare with searched section or no section specified *)
// 				RESULT := 1; (* section found *)
// 				OFFSET := i; (* take offset *)
// 				RUN := 0;
// 				state := 0;
// 			END_IF;
// 		ELSE
// 			pk := REF(KEY);
// 			pk^ := 0; (* KEY = '' *)
// 			RESULT := 11; (* key not found, section end - do not change offset *)
// 			RUN := 0;
// 			state := 0;
// 		END_IF;
// 	02:	(* key found *)
// 		IF RUN = 2 OR RUN = 3 THEN (* key preselected or report everything *)
// 			IF KEY = STR OR LEN(STR) = 0 THEN (* compare with searched key *)
// 				RESULT := 2; (* key found *)
// 				OFFSET := i; (* take offset *)
// 				RUN := 0;
// 				state := 0;
// 			END_IF;
// 		END_IF;
// 	03:	(* comment found *)
// 		OFFSET := i; (* take offset *)
// 		state := 0;
//
// 	05:	RESULT := 5; (* in progress *)
//
// 	10:	(* index out of range - end of buffer *)
// 		RESULT := 10; (* nothing found - end of data reached *)
// 		OFFSET := i; (* take offset *)
// 		RUN := 0;
// 		state := 0;
// 	END_CASE;
//
// 	(*####################  DEBUG-MESSAGE  ###################################*)
// 	(*IF _debug_enable THEN
// 		LOG_CL.NEW_MSG := 'IPF: intern Result ~1 , state ~2, step ~3 , offset ~4, run ~5';
// 		LOG_CL.PRINTF[1] := BYTE_TO_STRING(RESULT);
// 		LOG_CL.PRINTF[2] := BYTE_TO_STRING(state);
// 		LOG_CL.PRINTF[3] := INT_TO_STRING(step);
// 		LOG_CL.PRINTF[4] := UDINT_TO_STRING(OFFSET);
// 		LOG_CL.PRINTF[5] := BYTE_TO_STRING(RUN);
// 		LOG_MSG();
// 	END_IF;*)
// 	(*########################################################################*)
//
// END_IF;
//
// (*####################  DEBUG-MESSAGE  ###################################*)
// (*IF _debug_enable THEN
// 	IF step_last <> step THEN
// 		LOG_CL.NEW_MSG := 'IPB: Step: ~1';
// 		LOG_CL.PRINTF[1]  := INT_TO_STRING(step);
// 		LOG_MSG();
// 	END_IF;
// 	step_last := step;
// END_IF;*)
// (*########################################################################*)
// END_FUNCTION_BLOCK

// Commented out for beedance: it uses FLOAT_TO_REAL, which is commented out.
// FUNCTION_BLOCK IP2GEO
// VAR_IN_OUT
// 	IP_C : IP_C; (* IP_Control management structure *)
// 	S_BUF : NETWORK_BUFFER;
// 	R_BUF : NETWORK_BUFFER;
// 	GEO : IP2GEO_DATA;
// END_VAR
// VAR_INPUT
// 	IP : DWORD;
// 	ACTIVATE : BOOL;
// END_VAR
// VAR_OUTPUT
// 	BUSY : BOOL;
// 	DONE : BOOL;
// 	ERROR_C : DWORD;
// 	ERROR_T : BYTE;
// END_VAR
// VAR
// 	CTRL : XML_CONTROL;
// 	XML_READER : XML_READER;
// 	URL_DATA : url;
// 	DNS_CLIENT : DNS_CLIENT;
// 	HTTP_GET : HTTP_GET;
// 	last_state : BOOL;
// 	value_int :	INT;
// 	value_real : REAL;
// 	v_real : REAL;
// 	state : INT;
// END_VAR
// CASE state OF
//
// 00:
// 	IF ACTIVATE AND NOT last_state THEN
// 		state := 20;
// 		DONE := FALSE;
// 		BUSY := TRUE;
// 		ERROR_C := DWORD#0;
// 		ERROR_T := BYTE#0;
// 	END_IF;
//
// 20: (* URL for DNS AND HTTP-GET *)
// 	(* Example: http://ipinfodb.com/ip_query.php?ip=10.10.10.10 *)
// 	(* Example: http://ipinfodb.com/ip_query.php?timezone=true&IP=*)
// 	URL_DATA:=STRING_TO_URL(STR:='http://ipinfodb.com/ip_query.php?timezone=true&IP=',DEFAULT_PROTOCOL:='',DEFAULT_PATH:='');
//
// 	IF IP > DWORD#0 THEN
// 		URL_DATA.QUERY := CONCAT(URL_DATA.QUERY,IP4_TO_STRING(IP4:=IP));
// 	END_IF;
//
// 	state := 40;
//
// 40:
// 	IF DNS_CLIENT.DONE THEN
// 		state := 60;
// 	ELSIF (DNS_CLIENT.ERROR > DWORD#00) THEN
// 		(* error handling *)
// 		ERROR_C := DNS_CLIENT.ERROR;
// 		ERROR_T := BYTE#01;
// 		state := 100;
// 	END_IF;
//
// 60:
// 	IF HTTP_GET.DONE THEN
// 		state := 80;
// 		CTRL.START_POS := HTTP_GET.BODY_START;
// 		CTRL.STOP_POS := HTTP_GET.BODY_STOP;
// 		CTRL.COMMAND := WORD#2#10000000_00011000; (* ONLY TEXT AND ATTRIBUTE *)
// 		CTRL.WATCHDOG := T#1ms;
//
// 	ELSIF (HTTP_GET.ERROR > DWORD#00) THEN
// 		(* error handling *)
// 		ERROR_C := HTTP_GET.ERROR;
// 		ERROR_T := BYTE#02;
// 		state := 100;
// 	END_IF;
//
// 80:
// 	(* read XML data serially *)
// 	XML_READER(CTRL:=CTRL,BUF:=R_BUF.BUFFER);
// 	IF CTRL.TYP < 98 THEN (* evaluate only if not a watchdog pass *)
// 		(* perform automatic conversion to real and int *)
// 		value_int := 0;
// 		value_real := 0.0;
// 		IF LEN(CTRL.VALUE) <= 20 THEN
// 			v_real :=FLOAT_TO_REAL(FLT:=CTRL.VALUE);
// 			IF CHK_REAL(v_real) = 0 THEN (* !!! checks for a valid REAL value, otherwise TwinCAT crashes !!!!  *)
// 				value_real := v_real;
// 				value_int := REAL_TO_INT(value_real);
// 			END_IF;
// 		END_IF;
//
// 		CASE UINT_TO_INT(CTRL.COUNT) OF
//
// 		07: GEO.IP4 := IP4_DECODE(STR:=CTRL.VALUE); (* IP address *)
// 		10: GEO.STATE := 'OK' = CTRL.VALUE; (* STATUS *)
// 		13: GEO.COUNTRY_CODE := CTRL.VALUE; (* Country-Code *)
// 		16: GEO.COUNTRY_NAME := CTRL.VALUE; (* Country-Name *)
// 		19: GEO.REGION_CODE := CTRL.VALUE; (* Region-Code *)
// 		22: GEO.REGION_NAME := CTRL.VALUE; (* Region-Name *)
// 		25: GEO.CITY := CTRL.VALUE; (* City *)
// 		31: GEO.GEO_LATITUDE := value_real; (* Latitude *)
// 		34: GEO.GEO_LONGITUDE := value_real; (* Longitude *)
// 		37: GEO.TIME_ZONE_NAME := CTRL.VALUE; (* TimeZone Name *)
// 		40: GEO.GMT_OFFSET := value_int; (* GMT OFFSET in seconds *)
// 		43: GEO.IS_DST := value_int > 0; (* daylight saving time active *)
// 		END_CASE;
//
// 	ELSIF CTRL.TYP = 99 THEN (* EXIT - last element read *)
// 		DONE := TRUE;
// 		state := 100;
// 	END_IF;
//
// 100:
// 	(* UNLOCK HTTP DATA *)
// 	IF (NOT HTTP_GET.DONE) THEN
// 		state := 0;
// 		BUSY := FALSE;
// 		DONE := ERROR_T = BYTE#0;
// 	END_IF;
//
// END_CASE;
//
// (* ---------------- DNS --------------- *)
// DNS_CLIENT(	IP_C:=IP_C,
// 			S_BUF:=S_BUF,
// 			R_BUF:=R_BUF,
// 			DOMAIN:=URL_DATA.DOMAIN,
// 			IP4_DNS:=DWORD#00,
// 			ACTIVATE:=state=40 (* DNS Start *)
// 			);
//
// (* parameters not used, or not used directly *)
// (* 	DWORD :=DNS_CLIENT.IP4;
// 	BOOL  :=DNS_CLIENT.DONE;
// 	BYTE  :=DNS_CLIENT.ERROR; *)
// (* -------------------------------------*)
//
// (* ------------- HTTP_GET --------------- *)
// HTTP_GET(	IP_C:=IP_C,
// 			S_BUF:=S_BUF,
// 			R_BUF:=R_BUF,
// 			IP4:=DNS_CLIENT.IP4,
// 			GET:=state=60,
// 			MODE:=BYTE#2, (* HTTP 1.1 with persistent connection *)
// 			UNLOCK_BUF:=state=100,
// 			URL_DATA:=URL_DATA
// 			);
//
// (* parameters not used, or not used directly *)
// (*	STRING := HTTP_GET.HTTP_STATUS;
// 	UINT :=HTTP_GET.HEADER_START;
// 	UINT :=HTTP_GET.HEADER_STOP;
// 	UINT :=HTTP_GET.BODY_START;
// 	UINT :=HTTP_GET.BODY_STOP;
// 	BOOL :=HTTP_GET.DONE;
// 	BYTE :=HTTP_GET.ERROR;
// *)
// (* -------------------------------------*)
//
// last_state := ACTIVATE;
// END_FUNCTION_BLOCK

FUNCTION IP4_CHECK : BOOL
VAR_INPUT
	NIP : DWORD;
	LIP : DWORD;
	SM : DWORD;
END_VAR

IP4_CHECK := (NIP AND sm) = (LIP AND SM);
END_FUNCTION

FUNCTION IP4_DECODE : DWORD
VAR_INPUT
	str : STRING(15);
END_VAR
VAR
	pos: INT;
END_VAR

pos := FIND(str, '.');
WHILE pos > 0 DO
	IP4_DECODE := SHL(IP4_DECODE,8) OR STRING_TO_DWORD(LEFT(str,pos - 1));
	str := DELETE(str, pos, 1);
	pos := FIND(str, '.');
END_WHILE;
IP4_DECODE := SHL(IP4_DECODE,8) OR STRING_TO_DWORD(str);
END_FUNCTION

FUNCTION IP4_TO_STRING : STRING(15)
VAR_INPUT
	IP4 : DWORD;
END_VAR
VAR
	tmp : STRING(3);
END_VAR

(* mask bits AND INSERT AT given position *)
tmp := BYTE_TO_STRING(DWORD_TO_BYTE(IP4));
IP4_TO_STRING := CONCAT('...', tmp);
tmp := BYTE_TO_STRING(DWORD_TO_BYTE(SHR(IP4,8)));
IP4_TO_STRING := INSERT(IP4_TO_STRING, tmp, 2);
tmp := BYTE_TO_STRING(DWORD_TO_BYTE(SHR(IP4,16)));
IP4_TO_STRING := INSERT(IP4_TO_STRING, tmp, 1);
tmp := BYTE_TO_STRING(DWORD_TO_BYTE(SHR(IP4,24)));
IP4_TO_STRING := CONCAT(tmp, IP4_TO_STRING);
END_FUNCTION

FUNCTION_BLOCK IP_CONTROL
VAR_IN_OUT
	IP_C : IP_C; (* IP_Control management structure *)
	S_BUF : NETWORK_BUFFER; (* external send buffer *)
	R_BUF : NETWORK_BUFFER; (* external receive buffer *)
END_VAR
VAR_INPUT
	IP : DWORD; (* IP address *)
	PORT : WORD; (* port number *)
	TIME_OUT : TIME; (* monitoring time connect / send / receive *)
END_VAR
VAR
	c_time : UDINT; (* CONNECT time (time without a connection) *)
	s_time : UDINT; (* SEND time    (time since last data sent) *)
	r_time : UDINT; (* RECEIVE time (time since last data received) *)

	c_enable : BOOL; (* Connect: enable *)
	c_ip : DWORD; (* Connect: current IP address *)
	c_ip_str : STRING(15);
	c_port : WORD; (* Connect: current port number *)
	c_mode : BYTE; (* Connect: current mode UDP/TCP...... *)
	c_status : BYTE; (* Connect: Status (Errorcode) *)
	c_ready : BOOL; (* Connect: connection established *)
	c_ready_old : BOOL; (* Connect: last state of c_ready for edge evaluation *)

	s_total : INT; (* Send: total number of bytes to send *)
	s_cur_pos : INT; (* Send: current send position *)
	s_cur_size : INT; (* Send: current send size *)
	s_max_size : INT; (* Send: maximum telegram length for sending *)
	s_active : BOOL; (* Send: data sending is active *)
	s_status : BYTE; (* Send: Status (Errorcodes) *)
	s_ip_str : STRING(15);
	s_ip_exist : BOOL;

	r_status : BYTE; (* Receive: Status (Errorcodes) *)
	r_count : INT; (* Receive: number of received bytes *)
	r_offset : INT; (* Receive: current position in external receive buffer *)
	r_max_size : INT; (* Receive: size of the external receive buffer*)

	new_connection : BOOL; (* new connection parameters available *)
	tx : DWORD; (* last time value *)
	error_time : DWORD; (* current timeout value *)

	state: BYTE; (* step flag for connect *)
	bytes_received : DINT;
	udp_mode : BOOL;

	socket : T_HSOCKET;
	server : T_HSOCKET;
	fbCreate	: FB_SocketUdpCreate;
	fbConnect : FB_SocketConnect;
	fbClose : FB_SocketClose;
	fbSendTo : FB_SocketUdpSendTo;
	fbReceiveFrom : FB_SocketUdpReceiveFrom;
	fbSend : FB_SocketSend;
	fbReceive : FB_SocketReceive;
	fbListen : FB_SocketListen;
	fbAccept : FB_SocketAccept;
	nErrId : UDINT;
	Send_Busy : BOOL;
	Send_Error : BOOL;
	Send_ErrId : UDINT;

	IPCR : IP_CONTROL_RESET;

END_VAR

VAR CONSTANT
	STOP : BYTE := 0;
	UDP_INIT : BYTE:= 31;
	UDP_INIT_WAIT : BYTE:= 32;
	TC_INIT : BYTE := 51;
	TC_CONNECT : BYTE:= 52;
	TS_INIT : BYTE:= 53;
	TS_LISTEN_WAIT : BYTE:= 54;
	TS_ACCEPT : BYTE:= 55;
	TS_ACCEPT_WAIT : BYTE:= 56;
	C_CLOSE : BYTE := 190;
	C_CLOSE_WAIT : BYTE:= 191;
	C_CLOSE2 : BYTE := 192;
	C_CLOSE_WAIT2 : BYTE:= 193;
	C_WAIT : BYTE := 200;
	C_REC : BYTE := 210;
	C_REC_WAIT : BYTE := 211;
	C_SND : BYTE := 220;
	C_SND_WAIT1 : BYTE := 221;
	C_SND_WAIT2 : BYTE := 222;
END_VAR

(* on PLC reset or program download all old connections are closed *)
IPCR();
IF NOT IPCR.READY THEN RETURN; END_IF;

(*####################  DEBUG-MESSAGE  ###################################*)
(*########################################################################*)

(* read system time *)
tx := T_PLC_MS();

IF IP_C.C_PORT = 0 THEN
	IP_C.C_PORT := PORT; (* replace the given PORT with the configured PORT *)
END_IF;
IF IP_C.C_IP = 0 AND IP_C.C_MODE < 4 THEN
	IP_C.C_IP := IP; (* replace the given IP with the configured IP *)
END_IF;

new_connection := c_ip <> IP_C.C_IP OR c_mode <> IP_C.C_MODE OR c_port <> IP_C.C_PORT; (* new connection requested? *)
c_enable := IP_C.C_ENABLE AND NOT new_connection;

IF IP_C.C_ENABLE AND IP_C.ERROR = 0 AND state = STOP THEN (* enabled, no error, no socket open *)
	c_ip   := IP_C.C_IP;
	c_mode := IP_C.C_MODE;
	c_port := IP_C.C_PORT;
	c_ip_str := IP4_TO_STRING(c_ip);
	udp_mode := C_MODE.0; (* Mode 1,3,5 = udp *)

	error_time := TIME_TO_DWORD(MAX(T#200ms,TIME_OUT));
	IP_C.TIME_RESET := TRUE; (* reset all timers *)
	r_max_size := SIZEOF(R_BUF.BUFFER);
	s_max_size := SIZEOF(S_BUF.BUFFER);

	IF udp_mode THEN (* Mode: 1,3,5 = UDP CLIENT/SERVER *)
		state := UDP_INIT;
	ELSIF c_mode = 0 THEN (* Mode: 0 = TCP CLIENT *)
		state := TC_INIT;
	ELSE
		state := TS_INIT; (* Mode: 2,4 = TCP SERVER *)
	END_IF;

	IF c_mode < 5 THEN (* set receiver IP *)
		s_ip_str := c_ip_str;
		s_ip_exist := TRUE;
	ELSE
		s_ip_str := '';
		s_ip_exist := FALSE;
	END_IF;

    	(*####################  DEBUG-MESSAGE  ###################################*)
	(*########################################################################*)

END_IF;

(*####################  DEBUG-MESSAGE  ###################################*)
(*########################################################################*)

IF IP_C.TIME_RESET THEN (* reset all timers *)
	IP_C.TIME_RESET := FALSE; (* clear reset *)
	c_time := tx; (* reset connect timer *)
	s_time := tx; (* reset send timer *)
	r_time := tx; (* reset receive timer *)

	c_status := BYTE#0; (* reset last connect error *)
	s_status := BYTE#0; (* reset last send error *)
	r_status := BYTE#0; (* reset last receive error *)
END_IF;

(* ---------------------------------------------- *)

CASE state OF

UDP_INIT: (* UDP_CLIENT + SERVER *)

	fbCreate(bExecute := FALSE);
	fbCreate(	bExecute := TRUE , sSrvNetId := sSrvNetId, sLocalHost := sLocalHost, nLocalPort := SEL(c_mode = 1,c_port,0) , tTimeOut := TIME_OUT);
	fbCreate.bExecute := FALSE; (* presetting *)
	state := UDP_INIT_WAIT;

UDP_INIT_WAIT:
	fbCreate();
	IF NOT fbCreate.bBusy THEN
		IF NOT fbCreate.bError THEN
			socket := fbCreate.hSocket;
			c_ready := TRUE; (* Connected *)
			state := C_WAIT;
		ELSE
			c_status := 1; (* FB_SocketUdpCreate failed *)
			nErrId := fbCreate.nErrId;
			state := C_CLOSE;
		END_IF;
	END_IF;

(* ---------------------------------------------- *)
TC_INIT: (* TCP CLIENT (ACTIVE) *)
	fbConnect(bExecute := FALSE);
	fbConnect(bExecute := TRUE, sSrvNetId := sSrvNetId, sRemoteHost := c_ip_str, nRemotePort := c_port, tTimeout := TIME_OUT);
	fbConnect.bExecute := FALSE; (* presetting *)
	state := TC_CONNECT;

(* ---------------------------------------------- *)
TC_CONNECT:
	IF NOT c_enable OR c_status = 255 THEN (* not enabled or connect timeout *)
		state := C_CLOSE;
	END_IF;

	fbConnect();
	IF NOT fbConnect.bBusy THEN
		IF fbConnect.bError THEN
			nErrID := fbConnect.nErrId;
			state :=TC_INIT; (* try again *)
		ELSE
			socket := fbConnect.hSocket;
			c_ready := TRUE; (* Connected *)
			state := C_WAIT;
		END_IF;
	END_IF;
(* ---------------------------------------------- *)
TS_INIT: (* TCP SERVER (PASSIVE) *)
	fbListen(bExecute := FALSE);
	fbListen(bExecute := TRUE , sSrvNetId:= sSrvNetId , sLocalHost:= sLocalHost , nLocalPort:= c_port , tTimeout:= TIME_OUT);
	fbListen.bExecute := FALSE;
	state := TS_LISTEN_WAIT;
(* ---------------------------------------------- *)
TS_LISTEN_WAIT:
	fbListen();
	IF NOT fbListen.bBusy THEN
		IF fbListen.bError THEN
			c_status := 3; (* FB_SocketListen failed *)
			nErrID := fbListen.nErrId;
			state := C_CLOSE;
		ELSE
			server := fbListen.hListener;
			state := TS_ACCEPT;
		END_IF;
	END_IF;
(* ---------------------------------------------- *)
TS_ACCEPT:
	fbAccept(bExecute := FALSE);
	fbAccept(bExecute := TRUE, sSrvNetId := sSrvNetId, hListener := server, tTimeout := TIME_OUT);
	fbAccept.bExecute := FALSE;
	state := TS_ACCEPT_WAIT;
(* ---------------------------------------------- *)
TS_ACCEPT_WAIT:
	fbAccept();
	IF NOT fbAccept.bBusy THEN

		state := TS_ACCEPT; (* presetting  *)

		IF fbAccept.bError THEN
			c_status := 4; (* FB_SocketAccept failed *)
			nErrID := fbAccept.nErrId;
			state := C_CLOSE;
		ELSE (* no error *)
			IF fbAccept.bAccepted THEN
				socket := fbAccept.hSocket;
				IF socket.remoteAddr.sAddr  <> c_ip_str AND c_mode <> 4 THEN
					state := C_CLOSE; (* reject remote - close connection *)
				ELSE
					state := C_WAIT;
					c_ready := TRUE; (* Connected *)
				END_IF;
			END_IF; (* fbAccept.bAccepted *)
		END_IF; (* NOT fbAccept.bError *)
	END_IF; (*  NOT fbAccept.bBusy *)
(* ---------------------------------------------- *)
C_CLOSE:
	c_ready := FALSE;
	IF socket.handle > 0 THEN
		fbClose(bExecute := FALSE );
		fbClose(bExecute := TRUE, sSrvNetId := sSrvNetId,	hSocket := socket);
		fbClose.bExecute := FALSE;
		state := C_CLOSE_WAIT;
	ELSE
		state:= C_CLOSE2;
	END_IF;

C_CLOSE_WAIT:
	fbClose();
	IF NOT fbClose.bBusy THEN
		socket := TCPADS_NULL_HSOCKET; (* reset socket *)
		nErrId:= SEL(fbClose.bError,0,fbClose.nErrId);
		state:= C_CLOSE2;
	END_IF;

C_CLOSE2:
	IF server.handle > 0 THEN
		fbClose(bExecute := FALSE );
		fbClose(bExecute := TRUE, sSrvNetId := sSrvNetId,	hSocket := server);
		fbClose.bExecute := FALSE;
		state := C_CLOSE_WAIT2;
	ELSE
		state:= STOP;
	END_IF;

C_CLOSE_WAIT2:
	fbClose();
	IF NOT fbClose.bBusy THEN
		server := TCPADS_NULL_HSOCKET; (* reset socket *)
		nErrId:= SEL(fbClose.bError,0,fbClose.nErrId);
		state:= STOP;
	END_IF;

(* ---------------------------------------------- *)

C_WAIT: (* wait for request to close *)
	IF NOT c_enable OR NOT c_ready THEN
		state:= C_CLOSE;
	ELSIF S_BUF.SIZE > 0 AND IP_C.MAILBOX[2] = 0 AND s_ip_exist THEN
		state:= C_SND;
	ELSIF IP_C.MAILBOX[3] = 0 THEN
		state:= C_REC;
	END_IF;

(* ---------------------------------------------- *)

C_REC: (* receive data *)
	IF R_BUF.SIZE >= INT_TO_UINT(r_max_size) THEN
		R_BUF.SIZE := UINT#0;
		r_status := 254; (* receive buffer reset due to overflow *)
	END_IF;

	r_offset := SEL(udp_mode,UINT_TO_INT(R_BUF.SIZE),0);
	r_count := r_max_size - r_offset;
	bytes_received := 0;

	IF udp_mode THEN
		fbReceiveFrom(bExecute := FALSE );
		fbReceiveFrom(bExecute:= TRUE, sSrvNetId := sSrvNetId, hSocket:= socket, cbLen := r_count, pDest:= REF(R_BUF.BUFFER), tTimeout:= TIME_OUT);
		fbReceiveFrom.bExecute := FALSE; (* presetting *)
	ELSE
		fbReceive(bExecute:= FALSE);
		fbReceive(bExecute:= TRUE, sSrvNetId := sSrvNetId , hSocket:= socket , cbLen:= r_count, pDest:= REF(R_BUF.BUFFER[r_offset]) , tTimeout:= TIME_OUT);
		fbReceive.bExecute:= FALSE;
	END_IF;
	state := C_REC_WAIT;

C_REC_WAIT:
	IF udp_mode THEN
		fbReceiveFrom(); (* UDP Mode *)
		IF NOT fbReceiveFrom.bBusy THEN
			IF NOT fbReceiveFrom.bError THEN
				IF fbReceiveFrom.nRecBytes > 0 THEN
					IF c_mode <> BYTE#5 AND fbReceiveFrom.sRemoteHost  <> c_ip_str THEN
						R_BUF.SIZE := UINT#0;
					ELSE
						bytes_received := fbReceiveFrom.nRecBytes;
						IF NOT s_ip_exist THEN
							s_ip_str := fbReceiveFrom.sRemoteHost;
							s_ip_exist := TRUE;
						END_IF;
					END_IF;
				END_IF;
				state := C_WAIT;
			ELSIF fbReceiveFrom.nErrId = 16#80072746 THEN (* connection closed by remote *)
				c_status := 253;
				c_ready := FALSE;
				state := C_WAIT;
			ELSE
				nErrId := fbReceiveFrom.nErrId;
				state := C_WAIT;
			END_IF;
		END_IF;
	ELSE
		fbReceive(); (* TCP Mode *)
		IF NOT fbReceive.bBusy THEN
			IF NOT fbReceive.bError THEN
				IF fbReceive.nRecBytes > 0 THEN
					bytes_received := fbReceive.nRecBytes;
				END_IF;
			ELSIF fbReceive.nErrId = 16#8004 THEN (* connection closed by remote *)
				c_status := 253;
				c_ready := FALSE;
			ELSE
				nErrId := fbReceive.nErrId;
			END_IF;
			state := C_WAIT;
		END_IF;
	END_IF;

	IF bytes_received > 0 THEN
		r_time := tx; (* reset receive timer *)
		R_BUF.SIZE := INT_TO_UINT(r_offset + DINT_TO_UINT(bytes_received)); (* enter current buffer size *)
		IP_C.MAILBOX[1] := IP_C.MAILBOX[1] + 1; (* Receive Info *)
		IF IP_C.MAILBOX[1] = 0 THEN IP_C.MAILBOX[1] := 1; END_IF;
    		(*####################  DEBUG-MESSAGE  ###################################*)
		(*########################################################################*)
	END_IF;
